# B&R Automation Studio project NAELD004C00R10L518F00 (part 5)

#### Act_Main_P0201.st
```iecst
(** 2018-12-21 **)
ACTION Act_Main_P0201:

	//Machine Bitmap //def70
	IF p_tyNtParamCurr.eProjMag = LDMagDual AND p_tyNtParamCurr.sJobNo = '2023-0258A01' THEN //AT&S
		tyP0201OpsTravLifter.tyOps.tyBitmapMc.uiValueIdx	:= 441-70;
	ELSIF p_tyNtParamCurr.eProjMag = LDMagDual AND p_tyNtParamCurr.sJobNo = '2023-0276A01' THEN //clarion
		tyP0201OpsTravLifter.tyOps.tyBitmapMc.uiValueIdx	:= 471-70;
	ELSIF p_tyNtParamCurr.eProjMag = LDMagDual AND p_tyNtParamCurr.bMagAutoVerifyPrep = TRUE THEN
		tyP0201OpsTravLifter.tyOps.tyBitmapMc.uiValueIdx	:= 200;//270
	ELSIF p_tyNtParamCurr.eProjMag = LDMagDual AND p_tyNtParamCurr.bMagAutoVerifyPrep = FALSE THEN
		tyP0201OpsTravLifter.tyOps.tyBitmapMc.uiValueIdx	:= 200;
	ELSIF p_tyNtParamCurr.eProjMag = LDMagTriple AND p_tyNtParamCurr.bProjLifterMagPlatform THEN
		tyP0201OpsTravLifter.tyOps.tyBitmapMc.uiValueIdx	:= 398-70;
	ELSIF p_tyNtParamCurr.eProjMag = LDMagTriple AND p_tyNtParamCurr.bProjLifterMagPlatform = FALSE AND p_tyNtParamCurr.bProjCurtainSenPrep THEN
		tyP0201OpsTravLifter.tyOps.tyBitmapMc.uiValueIdx	:= 361-70;
	ELSIF p_tyNtParamCurr.eProjMag = LDMagTriple THEN
		tyP0201OpsTravLifter.tyOps.tyBitmapMc.uiValueIdx	:= 3;
	ELSIF p_tyNtParamCurr.eProjMag = LDMagQuadruple THEN
		tyP0201OpsTravLifter.tyOps.tyBitmapMc.uiValueIdx	:= 7;
		fUIInRtStatOff(ADR(tyP0201OpsTravLifter.tyOps.tyLyrProdRear.uiRtStat));

	ELSE
		tyP0201OpsTravLifter.tyOps.tyBitmapMc.uiValueIdx	:= 0;
		fUIInRtStatHide(ADR(tyP0201OpsTravLifter.tyOps.tyLyrProdRear.uiRtStat));
	END_IF

	IF p_tyNtParamCurr.eProjMag <> LDMagQuadruple THEN
		fUIInRtStatHide(ADR(tyP0201OpsTravLifter.tyOps.tyLyrProdRear.uiRtStat));
	END_IF
		//Display
	tyP0201OpsTravLifter.tyOps.tyBtnToptoBtm.uiRtStat.0	:= TRUE;
	IF p_tyNtParamCurr.bProjLaneBPrep = FALSE THEN
		fUIInRtStatHide(ADR(tyP0201OpsTravLifter.tyIOMonitor.tyBtnDSBB.uiRtStat));

		fUIInRtStatHide(ADR(tyP0201OpsTravLifter.tyIOMonitor.tyBtnDBAB.uiRtStat));
	END_IF

	IF p_tyNtParamCurr.bProjInletShutPrep = FALSE THEN
		fUIInRtStatHide(ADR(tyP0201OpsTravLifter.tyIOMonitor.tyBtnInletShutterCloseSen.uiRtStat));
		fUIInRtStatHide(ADR(tyP0201OpsTravLifter.tyIOMonitor.tyBtnInletShutterOpenSen.uiRtStat));
		fUIInRtStatHide(ADR(tyP0201OpsTravLifter.tyIOMonitor.tyBtnInShutterCloseCtrl.uiRtStat));
		fUIInRtStatHide(ADR(tyP0201OpsTravLifter.tyIOMonitor.tyBtnInShutterOpenCtrl.uiRtStat));
	END_IF
	IF p_tyNtParamCurr.bProjShutter2Prep = FALSE THEN
		fUIInRtStatHide(ADR(tyP0201OpsTravLifter.tyIOMonitor.tyBtnInletShutterCloseSen2.uiRtStat));
		fUIInRtStatHide(ADR(tyP0201OpsTravLifter.tyIOMonitor.tyBtnInletShutterOpenSen2.uiRtStat));
		fUIInRtStatHide(ADR(tyP0201OpsTravLifter.tyIOMonitor.tyBtnInShutterCloseCtrl2.uiRtStat));
		fUIInRtStatHide(ADR(tyP0201OpsTravLifter.tyIOMonitor.tyBtnInShutterOpenCtrl2.uiRtStat));
	END_IF
	IF p_tyNtParamCurr.bProjShutter3Prep = FALSE THEN
		fUIInRtStatHide(ADR(tyP0201OpsTravLifter.tyIOMonitor.tyBtnInletShutterCloseSen3.uiRtStat));
		fUIInRtStatHide(ADR(tyP0201OpsTravLifter.tyIOMonitor.tyBtnInletShutterOpenSen3.uiRtStat));
		fUIInRtStatHide(ADR(tyP0201OpsTravLifter.tyIOMonitor.tyBtnInShutterCloseCtrl3.uiRtStat));
		fUIInRtStatHide(ADR(tyP0201OpsTravLifter.tyIOMonitor.tyBtnInShutterOpenCtrl3.uiRtStat));
	END_IF

	IF p_tyNtParamCurr.bProjOutletShutPrep = FALSE THEN
		fUIInRtStatHide(ADR(tyP0201OpsTravLifter.tyIOMonitor.tyBtnOutletShutterCloseSen.uiRtStat));
		fUIInRtStatHide(ADR(tyP0201OpsTravLifter.tyIOMonitor.tyBtnOutletShutterOpenSen.uiRtStat));
		fUIInRtStatHide(ADR(tyP0201OpsTravLifter.tyIOMonitor.tyBtnOutShutterCloseCtrl.uiRtStat));
		fUIInRtStatHide(ADR(tyP0201OpsTravLifter.tyIOMonitor.tyBtnOutShutterOpenCtrl.uiRtStat));
	END_IF
	IF p_tyNtParamCurr.bProjOutShutter2Prep = FALSE THEN
		fUIInRtStatHide(ADR(tyP0201OpsTravLifter.tyIOMonitor.tyBtnOutletShutterCloseSen2.uiRtStat));
		fUIInRtStatHide(ADR(tyP0201OpsTravLifter.tyIOMonitor.tyBtnOutletShutterOpenSen2.uiRtStat));
		fUIInRtStatHide(ADR(tyP0201OpsTravLifter.tyIOMonitor.tyBtnOutShutterCloseCtrl2.uiRtStat));
		fUIInRtStatHide(ADR(tyP0201OpsTravLifter.tyIOMonitor.tyBtnOutShutterOpenCtrl2.uiRtStat));
	END_IF

	//Change Parameter
	IF p_tyNtParamCurr.bProjLaneBPrep THEN
		tyP0201OpsTravLifter.tyParam.tyDrpDnMcMode.usiValueMaxIdx	:= 2;
	ELSE
		tyP0201OpsTravLifter.tyParam.tyDrpDnMcMode.usiValueMaxIdx	:= 0;
	END_IF

	//Motorised puller
	tyP0201OpsTravLifter.tyOps.tyNumPshrOffset.uiRtStat := NOT p_tyNtParamCurr.bAWPusherPrep;
	tyP0201OpsTravLifter.tyOps.tyNumMtrPshrExtSpd.uiRtStat := NOT p_tyNtParamCurr.bProjMotorizedPullerPrep;
	tyP0201OpsTravLifter.tyOps.tyNumMtrPshrExtTorq.uiRtStat := NOT p_tyNtParamCurr.bProjMotorizedPullerPrep;
	tyP0201OpsTravLifter.tyParam.tyNumPshrOffset.uiRtStat := NOT p_tyNtParamCurr.bAWPusherPrep;
	tyP0201OpsTravLifter.tyParam.tyNumMtrPshrExtSpd.uiRtStat := NOT p_tyNtParamCurr.bProjMotorizedPullerPrep;
	tyP0201OpsTravLifter.tyParam.tyNumMtrPshrExtTorq.uiRtStat := NOT p_tyNtParamCurr.bProjMotorizedPullerPrep;

	//Digital Input Used
	IF p_tyNtParamCurr.tyDISettings.diSafetyRlySig = 0 THEN
		fUIInRtStatHide(ADR(tyP0201OpsTravLifter.tyIOMonitor.tyBtnSafetyRlySig.uiRtStat));
	END_IF

	IF p_tyNtParamCurr.tyDISettings.diEStopSig = 0 THEN
		fUIInRtStatHide(ADR(tyP0201OpsTravLifter.tyIOMonitor.tyBtnEStop.uiRtStat));
	END_IF

	IF p_tyNtParamCurr.tyDISettings.diCoverSWSig = 0 THEN
		fUIInRtStatHide(ADR(tyP0201OpsTravLifter.tyIOMonitor.tyBtnCoverSWSig.uiRtStat));
	END_IF

	IF p_tyNtParamCurr.tyDISettings.diDSBA = 0 THEN
		fUIInRtStatHide(ADR(tyP0201OpsTravLifter.tyIOMonitor.tyBtnDSBA.uiRtStat));
	END_IF

	IF p_tyNtParamCurr.tyDISettings.diDSBB = 0 THEN
		fUIInRtStatHide(ADR(tyP0201OpsTravLifter.tyIOMonitor.tyBtnDSBB.uiRtStat));
	END_IF

	IF p_tyNtParamCurr.tyDISettings.diPullerExtRS = 0 THEN
		fUIInRtStatHide(ADR(tyP0201OpsTravLifter.tyIOMonitor.tyBtnPullerExtRS.uiRtStat));
	END_IF

	IF p_tyNtParamCurr.tyDISettings.diPullerRetRS = 0 THEN
		fUIInRtStatHide(ADR(tyP0201OpsTravLifter.tyIOMonitor.tyBtnPullerRetRS.uiRtStat));
	END_IF

	IF p_tyNtParamCurr.tyDISettings.diPullerRotHmRS = 0 THEN
		fUIInRtStatHide(ADR(tyP0201OpsTravLifter.tyIOMonitor.tyBtnPullerRotCylHmRS.uiRtStat));
	END_IF

	IF p_tyNtParamCurr.tyDISettings.diPullerRotRmRS = 0 THEN
		fUIInRtStatHide(ADR(tyP0201OpsTravLifter.tyIOMonitor.tyBtnPullerRotCylRmRS.uiRtStat));
	END_IF

	IF p_tyNtParamCurr.tyDISettings.diConvLftSen = 0 THEN
		fUIInRtStatHide(ADR(tyP0201OpsTravLifter.tyIOMonitor.tyBtnConvLftSen.uiRtStat));
	END_IF

	IF p_tyNtParamCurr.tyDISettings.diConvRgtSen = 0 THEN
		fUIInRtStatHide(ADR(tyP0201OpsTravLifter.tyIOMonitor.tyBtnConvRgtSen.uiRtStat));
	END_IF

	IF p_tyNtParamCurr.tyDISettings.diLifterTimingBeltSen = 0 THEN
		fUIInRtStatHide(ADR(tyP0201OpsTravLifter.tyIOMonitor.tyBtnLifterTmBeltSen.uiRtStat));
	END_IF

	IF p_tyNtParamCurr.tyDISettings.diLifterSafetyLmtSW1 = 0 THEN
		fUIInRtStatHide(ADR(tyP0201OpsTravLifter.tyIOMonitor.tyBtnLifterSafetyLmtSw1.uiRtStat));
	END_IF

	IF p_tyNtParamCurr.tyDISettings.diLifterSafetyLmtSW2 = 0 THEN
		fUIInRtStatHide(ADR(tyP0201OpsTravLifter.tyIOMonitor.tyBtnLifterSafetyLmtSw2.uiRtStat));
	END_IF

	IF p_tyNtParamCurr.tyDISettings.diInShutterOpenRS = 0 THEN
		fUIInRtStatHide(ADR(tyP0201OpsTravLifter.tyIOMonitor.tyBtnInletShutterOpenSen.uiRtStat));
	END_IF

	IF p_tyNtParamCurr.tyDISettings.diInShutterCloseRS = 0 THEN
		fUIInRtStatHide(ADR(tyP0201OpsTravLifter.tyIOMonitor.tyBtnInletShutterCloseSen.uiRtStat));
	END_IF

	IF p_tyNtParamCurr.tyDISettings.diOutShutterOpenRS = 0 THEN
		fUIInRtStatHide(ADR(tyP0201OpsTravLifter.tyIOMonitor.tyBtnOutletShutterOpenSen.uiRtStat));
	END_IF

	IF p_tyNtParamCurr.tyDISettings.diOutShutterCloseRS = 0 THEN
		fUIInRtStatHide(ADR(tyP0201OpsTravLifter.tyIOMonitor.tyBtnOutletShutterCloseSen.uiRtStat));
	END_IF

	IF p_tyNtParamCurr.tyDISettings.diPullerAntiJam = 0 THEN
		fUIInRtStatHide(ADR(tyP0201OpsTravLifter.tyIOMonitor.tyBtnAntiJamSen.uiRtStat));
	END_IF
	tyP0201OpsTravLifter.tyIOMonitor.tyBtnMagWidthChk.uiRtStat := p_tyNtParamCurr.tyDISettings.diMagWidthChkSen =0;

	//Digital Output Selected
	IF p_tyNtParamCurr.tyDOSettings.diSafetyRlyRst = 0 THEN
		fUIInRtStatHide(ADR(tyP0201OpsTravLifter.tyIOMonitor.tyBtnSafetyRlyRst.uiRtStat));
	END_IF

	IF p_tyNtParamCurr.tyDOSettings.diTLGreen = 0 THEN
		fUIInRtStatHide(ADR(tyP0201OpsTravLifter.tyIOMonitor.tyBtnTLGreen.uiRtStat));
	END_IF

	IF p_tyNtParamCurr.tyDOSettings.diTLAmber = 0 THEN
		fUIInRtStatHide(ADR(tyP0201OpsTravLifter.tyIOMonitor.tyBtnTLAmber.uiRtStat));
	ELSE
		IF p_tyNtParamCurr.eTLBuzMode = TLBuzModSiemens_2Colour THEN
			tyP0201OpsTravLifter.tyIOMonitor.tyBtnTLAmber.usiTxtIdx := 333-253; //253 amber
		END_IF
	END_IF

	IF p_tyNtParamCurr.tyDOSettings.diTLRed = 0 THEN
		fUIInRtStatHide(ADR(tyP0201OpsTravLifter.tyIOMonitor.tyBtnTLRed.uiRtStat));
	END_IF

	IF p_tyNtParamCurr.tyDOSettings.diBuzzer = 0 THEN
		fUIInRtStatHide(ADR(tyP0201OpsTravLifter.tyIOMonitor.tyBtnBuzzer.uiRtStat));
	END_IF

	IF p_tyNtParamCurr.tyDOSettings.diDBAA = 0 THEN
		fUIInRtStatHide(ADR(tyP0201OpsTravLifter.tyIOMonitor.tyBtnDBAA.uiRtStat));
	END_IF

	IF p_tyNtParamCurr.tyDOSettings.diDBAB = 0 THEN
		fUIInRtStatHide(ADR(tyP0201OpsTravLifter.tyIOMonitor.tyBtnDBAB.uiRtStat));
	END_IF

	IF p_tyNtParamCurr.tyDOSettings.diPullerExtCtrl = 0 THEN
		fUIInRtStatHide(ADR(tyP0201OpsTravLifter.tyIOMonitor.tyBtnPullerExtCtrl.uiRtStat));
	END_IF

	IF p_tyNtParamCurr.tyDOSettings.diPullerRetCtrl = 0 THEN
		fUIInRtStatHide(ADR(tyP0201OpsTravLifter.tyIOMonitor.tyBtnPullerRetCtrl.uiRtStat));
	END_IF

	IF p_tyNtParamCurr.tyDOSettings.diRotPullerCtrl = 0 THEN
		fUIInRtStatHide(ADR(tyP0201OpsTravLifter.tyIOMonitor.tyBtnRotPullerCtrl.uiRtStat));
	END_IF

	IF p_tyNtParamCurr.tyDOSettings.diInShutterOpenCtrl = 0 THEN
		fUIInRtStatHide(ADR(tyP0201OpsTravLifter.tyIOMonitor.tyBtnInShutterOpenCtrl.uiRtStat));
	END_IF

	IF p_tyNtParamCurr.tyDOSettings.diInShutterCloseCtrl = 0 THEN
		fUIInRtStatHide(ADR(tyP0201OpsTravLifter.tyIOMonitor.tyBtnInShutterCloseCtrl.uiRtStat));
	END_IF

	IF p_tyNtParamCurr.tyDOSettings.diOutShutterOpenCtrl = 0 THEN
		fUIInRtStatHide(ADR(tyP0201OpsTravLifter.tyIOMonitor.tyBtnOutShutterOpenCtrl.uiRtStat));
	END_IF

	IF p_tyNtParamCurr.tyDOSettings.diOutShutterCloseCtrl = 0 THEN
		fUIInRtStatHide(ADR(tyP0201OpsTravLifter.tyIOMonitor.tyBtnOutShutterCloseCtrl.uiRtStat));
	END_IF

	IF p_tyNtParamCurr.tyDOSettings.diPullConvMtrOn = 0 THEN
		fUIInRtStatHide(ADR(tyP0201OpsTravLifter.tyIOMonitor.tyBtnPullerConvMtrOn.uiRtStat));
	END_IF

	tyP0201OpsTravLifter.tyIOMonitor.tyBtnConvClrSen.uiRtStat := 	p_tyNtParamCurr.tyDISettings.diConvClrSen =0;
	tyP0201OpsTravLifter.tyIOMonitor.tyBtnUnlockSigDS.uiRtStat := 	p_tyNtParamCurr.tyDISettings.diDSUnlockCoverSig =0;
	tyP0201OpsTravLifter.tyIOMonitor.tyBtnSafetySigDS.uiRtStat := 	p_tyNtParamCurr.tyDISettings.diDSSafetySig =0;
	tyP0201OpsTravLifter.tyIOMonitor.tyBtnSftySglToUSDS.uiRtStat := 	p_tyNtParamCurr.tyDOSettings.diMcSafetySigToDS =0;

//	IF p_tyNtParamCurr.bLFProdWidth2Prep THEN
//		fUIInRtStatOff(ADR(tyP0201OpsTravLifter.tyOps.tyNumWidth2.uiRtStat));
//		fUIInRtStatHide(ADR(tyP0201OpsTravLifter.tyOps.tyNumWidth.uiRtStat));
//	ELSE
//		fUIInRtStatHide(ADR(tyP0201OpsTravLifter.tyOps.tyNumWidth2.uiRtStat));
//		fUIInRtStatOff(ADR(tyP0201OpsTravLifter.tyOps.tyNumWidth.uiRtStat));
//	END_IF
//
//	IF p_tyNtParamCurr.eProjMag = LDMagQuadruple THEN
//		fUIInRtStatOff(ADR(tyP0201OpsTravLifter.tyOps.tyNumWidth2.uiRtStat));
//		fUIInRtStatHide(ADR(tyP0201OpsTravLifter.tyOps.tyNumWidth.uiRtStat));
//	ELSE
		fUIInRtStatHide(ADR(tyP0201OpsTravLifter.tyOps.tyNumWidth2.uiRtStat));
		fUIInRtStatOff(ADR(tyP0201OpsTravLifter.tyOps.tyNumWidth.uiRtStat));
//	END_IF

END_ACTION
```

#### Act_Main_P0202.st
```iecst
(** 2018-12-21 **)
ACTION Act_Main_P0202:

	//Machine Bitmap//71

	IF p_tyNtParamCurr.eProjMag = LDMagDual AND p_tyNtParamCurr.sJobNo = '2023-0258A01' THEN //AT&S
		tyP0202OpsMag1.tyOps.tyBitmapMc.uiValueIdx	:= 442-71;
	ELSIF p_tyNtParamCurr.eProjMag = LDMagDual AND p_tyNtParamCurr.sJobNo = '2023-0276A01' THEN //clarion (RL)
		tyP0202OpsMag1.tyOps.tyBitmapMc.uiValueIdx	:= 472-71;
	ELSIF p_tyNtParamCurr.eProjMag = LDMagDual AND p_tyNtParamCurr.bMagAutoVerifyPrep = TRUE THEN
		tyP0202OpsMag1.tyOps.tyBitmapMc.uiValueIdx	:= 200;
	ELSIF p_tyNtParamCurr.eProjMag = LDMagDual AND p_tyNtParamCurr.bMagAutoVerifyPrep = FALSE THEN
		tyP0202OpsMag1.tyOps.tyBitmapMc.uiValueIdx	:= 200;
	ELSIF p_tyNtParamCurr.eProjMag = LDMagTriple AND p_tyNtParamCurr.bProjLifterMagPlatform THEN
		tyP0202OpsMag1.tyOps.tyBitmapMc.uiValueIdx	:= 399-71;
	ELSIF p_tyNtParamCurr.eProjMag = LDMagTriple AND p_tyNtParamCurr.bProjLifterMagPlatform =FALSE AND p_tyNtParamCurr.bProjCurtainSenPrep THEN
		tyP0202OpsMag1.tyOps.tyBitmapMc.uiValueIdx	:= 362-71;
	ELSIF p_tyNtParamCurr.eProjMag = LDMagTriple THEN
		tyP0202OpsMag1.tyOps.tyBitmapMc.uiValueIdx	:= 3;
	ELSIF p_tyNtParamCurr.eProjMag = LDMagQuadruple THEN
		tyP0202OpsMag1.tyOps.tyBitmapMc.uiValueIdx	:= 7;
	ELSE
		tyP0202OpsMag1.tyOps.tyBitmapMc.uiValueIdx	:= 0;
	END_IF

	//AIV
	tyP0202OpsMag1.tyOps.tyTxtLblAIV.uiRtStat.0		:= NOT p_tyNtParamCurr.bProjAGVPrep;
	tyP0202OpsMag1.tyOps.tyBtnAIVWifi.uiRtStat.0	:= NOT p_tyNtParamCurr.bProjAGVPrep;
	tyP0202OpsMag1.tyOps.tyBtnChgMag.uiRtStat.0		:= NOT(p_tyNtParamCurr.bProjAGVPrep AND p_tyNtParamCurr.bProjBtnInsertRmvMag);
	tyP0202OpsMag1.tyOps.tyBitmapChgMag.uiRtStat.0	:= NOT(p_tyNtParamCurr.bProjAGVPrep AND p_tyNtParamCurr.bProjBtnInsertRmvMag);

	//Motorized puller
	tyP0202OpsMag1.tyParam.tyNumPshrOffset.uiRtStat := NOT p_tyNtParamCurr.bAWPusherPrep;
	tyP0202OpsMag1.tyParam.tyNumMtrPshrExtSpd.uiRtStat := NOT p_tyNtParamCurr.bProjMotorizedPullerPrep;
	tyP0202OpsMag1.tyParam.tyNumMtrPshrExtTorq.uiRtStat := NOT p_tyNtParamCurr.bProjMotorizedPullerPrep;

	//Display
	IF p_tyNtParamCurr.bProjLaneBPrep = FALSE THEN
		fUIInRtStatHide(ADR(tyP0202OpsMag1.tyIOMonitor.tyBtnDSBB.uiRtStat));

		fUIInRtStatHide(ADR(tyP0202OpsMag1.tyIOMonitor.tyBtnDBAB.uiRtStat));
	END_IF
	tyP0202OpsMag1.tyOps.tyBtnToptoBtm.uiRtStat.0	:= TRUE;
	//Change Parameter
	IF p_tyNtParamCurr.bProjLaneBPrep THEN
		tyP0202OpsMag1.tyParam.tyDrpDnMcMode.usiValueMaxIdx	:= 2;
	ELSE
		tyP0202OpsMag1.tyParam.tyDrpDnMcMode.usiValueMaxIdx	:= 0;
	END_IF

	//Digital Input Used
	IF p_tyNtParamCurr.tyDISettings.diSafetyRlySig = 0 THEN
		fUIInRtStatHide(ADR(tyP0202OpsMag1.tyIOMonitor.tyBtnSafetyRlySig.uiRtStat));
	END_IF

	IF p_tyNtParamCurr.tyDISettings.diEStopSig = 0 THEN
		fUIInRtStatHide(ADR(tyP0202OpsMag1.tyIOMonitor.tyBtnEStop.uiRtStat));
	END_IF

	IF p_tyNtParamCurr.tyDISettings.diCoverSWSig = 0 THEN
		fUIInRtStatHide(ADR(tyP0202OpsMag1.tyIOMonitor.tyBtnCoverSWSig.uiRtStat));
	END_IF

	IF p_tyNtParamCurr.tyDISettings.diDSBA = 0 THEN
		fUIInRtStatHide(ADR(tyP0202OpsMag1.tyIOMonitor.tyBtnDSBA.uiRtStat));
	END_IF

	IF p_tyNtParamCurr.tyDISettings.diDSBB = 0 THEN
		fUIInRtStatHide(ADR(tyP0202OpsMag1.tyIOMonitor.tyBtnDSBB.uiRtStat));
	END_IF

	IF p_tyNtParamCurr.tyDISettings.diMag1FixedClampRS = 0 THEN
		fUIInRtStatHide(ADR(tyP0202OpsMag1.tyIOMonitor.tyBtnMag1FixedClmpRS.uiRtStat));
	END_IF

	IF p_tyNtParamCurr.tyDISettings.diMag1FixedUnclampRS = 0 THEN
		fUIInRtStatHide(ADR(tyP0202OpsMag1.tyIOMonitor.tyBtnMag1FixedUnclmpRS.uiRtStat));
	END_IF

	IF p_tyNtParamCurr.tyDISettings.diMag1RemoteClampRS = 0 THEN
		fUIInRtStatHide(ADR(tyP0202OpsMag1.tyIOMonitor.tyBtnMag1RmtClmpRS.uiRtStat));
	END_IF

	IF p_tyNtParamCurr.tyDISettings.diMag1RemoteUnclampRS = 0 THEN
		fUIInRtStatHide(ADR(tyP0202OpsMag1.tyIOMonitor.tyBtnMag1RmtUnclmpRS.uiRtStat));
	END_IF

	IF p_tyNtParamCurr.tyDISettings.diMagConvEntSen1 = 0 THEN
		fUIInRtStatHide(ADR(tyP0202OpsMag1.tyIOMonitor.tyBtnMag1ConvEntrySen.uiRtStat));
	END_IF

	IF p_tyNtParamCurr.tyDISettings.diMagPresentSen1 = 0 THEN
		fUIInRtStatHide(ADR(tyP0202OpsMag1.tyIOMonitor.tyBtnMag1PresentSen.uiRtStat));
	END_IF

	IF p_tyNtParamCurr.tyDISettings.diMag1AGVInPosSen1 = 0 THEN
		fUIInRtStatHide(ADR(tyP0202OpsMag1.tyIOMonitor.tyBtnMag1AIVInPosSen1.uiRtStat));
	END_IF

	IF p_tyNtParamCurr.tyDISettings.diMag1AGVInPosSen2 = 0 THEN
		fUIInRtStatHide(ADR(tyP0202OpsMag1.tyIOMonitor.tyBtnMag1AIVInPosSen2.uiRtStat));
	END_IF

	IF p_tyNtParamCurr.tyDISettings.diMag1OrientChkSen1 = 0 THEN
		fUIInRtStatHide(ADR(tyP0202OpsMag1.tyIOMonitor.tyBtnMag1OrientationChkSen1.uiRtStat));
	END_IF

	IF p_tyNtParamCurr.tyDISettings.diMag1OrientChkSen2 = 0 THEN
		fUIInRtStatHide(ADR(tyP0202OpsMag1.tyIOMonitor.tyBtnMag1OrientationChkSen2.uiRtStat));
	END_IF

	tyP0202OpsMag1.tyIOMonitor.tyBtnMagDetSen.uiRtStat.0			:= p_tyNtParamCurr.tyDISettings.diMag1FixedSideDetect = 0;
	tyP0202OpsMag1.tyIOMonitor.tyBtnTrllyExtRS.uiRtStat.0			:= p_tyNtParamCurr.tyDISettings.diTrolleyExtRS1 = 0;
	tyP0202OpsMag1.tyIOMonitor.tyBtnTrllyPresentSen.uiRtStat.0		:= p_tyNtParamCurr.tyDISettings.diTrolleyPreSen1 = 0;
	tyP0202OpsMag1.tyIOMonitor.tyBtnSltLckSen.uiRtStat.0			:= p_tyNtParamCurr.tyDISettings.diSlotLckSenMag1 = 0;

	//Digital Output Selected
	IF p_tyNtParamCurr.tyDOSettings.diSafetyRlyRst = 0 THEN
		fUIInRtStatHide(ADR(tyP0202OpsMag1.tyIOMonitor.tyBtnSafetyRlyRst.uiRtStat));
	END_IF

	IF p_tyNtParamCurr.tyDOSettings.diTLGreen = 0 THEN
		fUIInRtStatHide(ADR(tyP0202OpsMag1.tyIOMonitor.tyBtnTLGreen.uiRtStat));
	END_IF

	IF p_tyNtParamCurr.tyDOSettings.diTLAmber = 0 THEN
		fUIInRtStatHide(ADR(tyP0202OpsMag1.tyIOMonitor.tyBtnTLAmber.uiRtStat));
	ELSE
		IF p_tyNtParamCurr.eTLBuzMode = TLBuzModSiemens_2Colour THEN
			tyP0202OpsMag1.tyIOMonitor.tyBtnTLAmber.usiTxtIdx := 333-253; //253 amber
		END_IF
	END_IF

	IF p_tyNtParamCurr.tyDOSettings.diTLRed = 0 THEN
		fUIInRtStatHide(ADR(tyP0202OpsMag1.tyIOMonitor.tyBtnTLRed.uiRtStat));
	END_IF

	IF p_tyNtParamCurr.tyDOSettings.diBuzzer = 0 THEN
		fUIInRtStatHide(ADR(tyP0202OpsMag1.tyIOMonitor.tyBtnBuzzer.uiRtStat));
	END_IF

	IF p_tyNtParamCurr.tyDOSettings.diDBAA = 0 THEN
		fUIInRtStatHide(ADR(tyP0202OpsMag1.tyIOMonitor.tyBtnDBAA.uiRtStat));
	END_IF

	IF p_tyNtParamCurr.tyDOSettings.diDBAB = 0 THEN
		fUIInRtStatHide(ADR(tyP0202OpsMag1.tyIOMonitor.tyBtnDBAB.uiRtStat));
	END_IF

	IF p_tyNtParamCurr.tyDOSettings.diMag1FixedClampCtrl = 0 THEN
		fUIInRtStatHide(ADR(tyP0202OpsMag1.tyIOMonitor.tyBtnMag1FixedClampCtrl.uiRtStat));
	END_IF

	IF p_tyNtParamCurr.tyDOSettings.diMag1FixedClampOpenCtrl = 0 THEN //KS
		fUIInRtStatHide(ADR(tyP0202OpsMag1.tyIOMonitor.tyBtnMag1FixedClampCtrl.uiRtStat));
	END_IF

	IF p_tyNtParamCurr.tyDOSettings.diMag1RemoteClampCtrl = 0 THEN
		fUIInRtStatHide(ADR(tyP0202OpsMag1.tyIOMonitor.tyBtnMag1RemoteClampCtrl.uiRtStat));
	END_IF

	IF p_tyNtParamCurr.tyDOSettings.diMag1RemoteClampOpenCtrl = 0 THEN //KS
		fUIInRtStatHide(ADR(tyP0202OpsMag1.tyIOMonitor.tyBtnMag1RemoteClampCtrl.uiRtStat));
	END_IF

	IF p_tyNtParamCurr.tyDOSettings.diMag1ConvMtrIn = 0 THEN
		fUIInRtStatHide(ADR(tyP0202OpsMag1.tyIOMonitor.tyBtnMag1ConvMtrIn.uiRtStat));
	END_IF

	IF p_tyNtParamCurr.tyDOSettings.diMag1ConvMtrOut = 0 THEN
		fUIInRtStatHide(ADR(tyP0202OpsMag1.tyIOMonitor.tyBtnMag1ConvMtrOut.uiRtStat));
	END_IF
	tyP0202OpsMag1.tyIOMonitor.tyBtnTrllyExtCtrl.uiRtStat.0			:= p_tyNtParamCurr.tyDOSettings.diTrolleyLckCtrl1 = 0;

	tyP0202OpsMag1.tyIOMonitor.tyBtnMagSelClampCtrl.uiRtStat.0		:= NOT p_tyNtParamCurr.bMagAutoVerifyPrep;
	tyP0202OpsMag1.tyIOMonitor.tyBtnHeightSen.uiRtStat.0			:= NOT (p_tyNtParamCurr.bMagAutoVerifyPrep OR p_tyNtParamCurr.bProjMagHeightChkPrep);
	tyP0202OpsMag1.tyIOMonitor.tyBtnCAB717Sen.uiRtStat.0			:= NOT p_tyNtParamCurr.bMagAutoVerifyPrep;
	tyP0202OpsMag1.tyIOMonitor.tyBtnMagLargeSen.uiRtStat.0			:= NOT p_tyNtParamCurr.bMagAutoVerifyPrep;
	tyP0202OpsMag1.tyIOMonitor.tyBtnMagSmallSen.uiRtStat.0			:= NOT p_tyNtParamCurr.bMagAutoVerifyPrep;
	tyP0202OpsMag1.tyIOMonitor.tyBtnSelUnclampRS.uiRtStat.0			:= NOT p_tyNtParamCurr.bMagAutoVerifyPrep;

//	IF p_tyNtParamCurr.eProjMag = LDMagQuadruple THEN
//		fUIInRtStatOff(ADR(tyP0202OpsMag1.tyOps.tyNumWidth2.uiRtStat));
//		fUIInRtStatHide(ADR(tyP0202OpsMag1.tyOps.tyNumWidth.uiRtStat));
//	ELSE
		fUIInRtStatHide(ADR(tyP0202OpsMag1.tyOps.tyNumWidth2.uiRtStat));
		fUIInRtStatOff(ADR(tyP0202OpsMag1.tyOps.tyNumWidth.uiRtStat));
//	END_IF

	tyP0202OpsMag1.tyOps.tyBtnUnloadMag.uiRtStat.0 := NOT p_tyNtParamCurr.bProjLifterMagPlatform;
	tyP0202OpsMag1.tyOps.tyBitmapUnloadMag.uiRtStat.0 := NOT p_tyNtParamCurr.bProjLifterMagPlatform;
	tyP0202OpsMag1.tyOps.tyBtnChgMag.uiRtStat.0 := p_tyNtParamCurr.bProjLifterMagPlatform;

END_ACTION
```

#### Act_Main_P0203.st
```iecst
(** 2018-12-21 **)
ACTION Act_Main_P0203:

	//Machine Bitmap//72
	IF p_tyNtParamCurr.eProjMag = LDMagDual AND p_tyNtParamCurr.sJobNo = '2023-0258A01' THEN //AT&S
		tyP0203OpsMag2.tyOps.tyBitmapMc.uiValueIdx	:= 443-72;
	ELSIF p_tyNtParamCurr.eProjMag = LDMagDual AND p_tyNtParamCurr.sJobNo = '2023-0276A01' THEN //clarion (RL)
		tyP0203OpsMag2.tyOps.tyBitmapMc.uiValueIdx	:= 473-72;
	ELSIF p_tyNtParamCurr.eProjMag = LDMagDual AND p_tyNtParamCurr.bMagAutoVerifyPrep = TRUE THEN
		tyP0203OpsMag2.tyOps.tyBitmapMc.uiValueIdx	:= 200;
	ELSIF p_tyNtParamCurr.eProjMag = LDMagDual AND p_tyNtParamCurr.bMagAutoVerifyPrep = FALSE THEN
		tyP0203OpsMag2.tyOps.tyBitmapMc.uiValueIdx	:= 200;
	ELSIF p_tyNtParamCurr.eProjMag = LDMagTriple AND p_tyNtParamCurr.bProjLifterMagPlatform THEN
		tyP0203OpsMag2.tyOps.tyBitmapMc.uiValueIdx	:= 400-72;
	ELSIF p_tyNtParamCurr.eProjMag = LDMagTriple AND p_tyNtParamCurr.bProjLifterMagPlatform =FALSE AND p_tyNtParamCurr.bProjCurtainSenPrep THEN
		tyP0203OpsMag2.tyOps.tyBitmapMc.uiValueIdx	:= 363-72;
	ELSIF p_tyNtParamCurr.eProjMag = LDMagTriple THEN
		tyP0203OpsMag2.tyOps.tyBitmapMc.uiValueIdx	:= 3;
	ELSIF p_tyNtParamCurr.eProjMag = LDMagQuadruple THEN
		tyP0203OpsMag2.tyOps.tyBitmapMc.uiValueIdx	:= 7;
	ELSE
		tyP0203OpsMag2.tyOps.tyBitmapMc.uiValueIdx	:= 0;
	END_IF

	//AIV
	tyP0203OpsMag2.tyOps.tyTxtLblAIV.uiRtStat.0		:= NOT p_tyNtParamCurr.bProjAGVPrep;
	tyP0203OpsMag2.tyOps.tyBtnAIVWifi.uiRtStat.0	:= NOT p_tyNtParamCurr.bProjAGVPrep;
	tyP0203OpsMag2.tyOps.tyBtnChgMag.uiRtStat.0		:= NOT(p_tyNtParamCurr.bProjAGVPrep AND p_tyNtParamCurr.bProjBtnInsertRmvMag);
	tyP0203OpsMag2.tyOps.tyBitmapChgMag.uiRtStat.0	:= NOT(p_tyNtParamCurr.bProjAGVPrep AND p_tyNtParamCurr.bProjBtnInsertRmvMag);

	//Motorized puller
	tyP0203OpsMag2.tyParam.tyNumPshrOffset.uiRtStat := NOT p_tyNtParamCurr.bAWPusherPrep;
	tyP0203OpsMag2.tyParam.tyNumMtrPshrExtSpd.uiRtStat := NOT p_tyNtParamCurr.bProjMotorizedPullerPrep;
	tyP0203OpsMag2.tyParam.tyNumMtrPshrExtTorq.uiRtStat := NOT p_tyNtParamCurr.bProjMotorizedPullerPrep;

	//Display
	IF p_tyNtParamCurr.bProjLaneBPrep = FALSE THEN
		fUIInRtStatHide(ADR(tyP0203OpsMag2.tyIOMonitor.tyBtnDSBB.uiRtStat));

		fUIInRtStatHide(ADR(tyP0203OpsMag2.tyIOMonitor.tyBtnDBAB.uiRtStat));
	END_IF
	tyP0203OpsMag2.tyOps.tyBtnToptoBtm.uiRtStat.0	:= TRUE;
	//Change Parameter
	IF p_tyNtParamCurr.bProjLaneBPrep THEN
		tyP0203OpsMag2.tyParam.tyDrpDnMcMode.usiValueMaxIdx	:= 2;
	ELSE
		tyP0203OpsMag2.tyParam.tyDrpDnMcMode.usiValueMaxIdx	:= 0;
	END_IF

	//Digital Input Used
	IF p_tyNtParamCurr.tyDISettings.diSafetyRlySig = 0 THEN
		fUIInRtStatHide(ADR(tyP0203OpsMag2.tyIOMonitor.tyBtnSafetyRlySig.uiRtStat));
	END_IF

	IF p_tyNtParamCurr.tyDISettings.diEStopSig = 0 THEN
		fUIInRtStatHide(ADR(tyP0203OpsMag2.tyIOMonitor.tyBtnEStop.uiRtStat));
	END_IF

	IF p_tyNtParamCurr.tyDISettings.diCoverSWSig = 0 THEN
		fUIInRtStatHide(ADR(tyP0203OpsMag2.tyIOMonitor.tyBtnCoverSWSig.uiRtStat));
	END_IF

	IF p_tyNtParamCurr.tyDISettings.diDSBA = 0 THEN
		fUIInRtStatHide(ADR(tyP0203OpsMag2.tyIOMonitor.tyBtnDSBA.uiRtStat));
	END_IF

	IF p_tyNtParamCurr.tyDISettings.diDSBB = 0 THEN
		fUIInRtStatHide(ADR(tyP0203OpsMag2.tyIOMonitor.tyBtnDSBB.uiRtStat));
	END_IF

	IF p_tyNtParamCurr.tyDISettings.diMag2FixedClampRS = 0 THEN
		fUIInRtStatHide(ADR(tyP0203OpsMag2.tyIOMonitor.tyBtnMag2FixedClmpRS.uiRtStat));
	END_IF

	IF p_tyNtParamCurr.tyDISettings.diMag2FixedUnclampRS = 0 THEN
		fUIInRtStatHide(ADR(tyP0203OpsMag2.tyIOMonitor.tyBtnMag2FixedUnclmpRS.uiRtStat));
	END_IF

	IF p_tyNtParamCurr.tyDISettings.diMag2RemoteClampRS = 0 THEN
		fUIInRtStatHide(ADR(tyP0203OpsMag2.tyIOMonitor.tyBtnMag2RmtClmpRS.uiRtStat));
	END_IF

	IF p_tyNtParamCurr.tyDISettings.diMag2RemoteUnclampRS = 0 THEN
		fUIInRtStatHide(ADR(tyP0203OpsMag2.tyIOMonitor.tyBtnMag2RmtUnclmpRS.uiRtStat));
	END_IF

	IF p_tyNtParamCurr.tyDISettings.diMagConvEntSen2 = 0 THEN
		fUIInRtStatHide(ADR(tyP0203OpsMag2.tyIOMonitor.tyBtnMag2ConvEntrySen.uiRtStat));
	END_IF

	IF p_tyNtParamCurr.tyDISettings.diMagPresentSen2 = 0 THEN
		fUIInRtStatHide(ADR(tyP0203OpsMag2.tyIOMonitor.tyBtnMag2PresentSen.uiRtStat));
	END_IF

	IF p_tyNtParamCurr.tyDISettings.diMag2AGVInPosSen1 = 0 THEN
		fUIInRtStatHide(ADR(tyP0203OpsMag2.tyIOMonitor.tyBtnMag2AIVInPosSen1.uiRtStat));
	END_IF

	IF p_tyNtParamCurr.tyDISettings.diMag2AGVInPosSen2 = 0 THEN
		fUIInRtStatHide(ADR(tyP0203OpsMag2.tyIOMonitor.tyBtnMag2AIVInPosSen2.uiRtStat));
	END_IF

	IF p_tyNtParamCurr.tyDISettings.diMag1OrientChkSen1 = 0 THEN
		fUIInRtStatHide(ADR(tyP0203OpsMag2.tyIOMonitor.tyBtnMag2OrientationChkSen1.uiRtStat));
	END_IF

	IF p_tyNtParamCurr.tyDISettings.diMag2OrientChkSen2 = 0 THEN
		fUIInRtStatHide(ADR(tyP0203OpsMag2.tyIOMonitor.tyBtnMag2OrientationChkSen2.uiRtStat));
	END_IF
	tyP0203OpsMag2.tyIOMonitor.tyBtnMagDetSen.uiRtStat.0			:= p_tyNtParamCurr.tyDISettings.diMag2FixedSideDetect = 0;
	tyP0203OpsMag2.tyIOMonitor.tyBtnTrllyExtRS.uiRtStat.0			:= p_tyNtParamCurr.tyDISettings.diTrolleyExtRS2 = 0;
	tyP0203OpsMag2.tyIOMonitor.tyBtnTrllyPresentSen.uiRtStat.0		:= p_tyNtParamCurr.tyDISettings.diTrolleyPreSen2 = 0;
	tyP0203OpsMag2.tyIOMonitor.tyBtnSltLckSen.uiRtStat.0			:= p_tyNtParamCurr.tyDISettings.diSlotLckSenMag2 = 0;

	//Digital Output Selected
	IF p_tyNtParamCurr.tyDOSettings.diSafetyRlyRst = 0 THEN
		fUIInRtStatHide(ADR(tyP0203OpsMag2.tyIOMonitor.tyBtnSafetyRlyRst.uiRtStat));
	END_IF

	IF p_tyNtParamCurr.tyDOSettings.diTLGreen = 0 THEN
		fUIInRtStatHide(ADR(tyP0203OpsMag2.tyIOMonitor.tyBtnTLGreen.uiRtStat));
	END_IF

	IF p_tyNtParamCurr.tyDOSettings.diTLAmber = 0 THEN
		fUIInRtStatHide(ADR(tyP0203OpsMag2.tyIOMonitor.tyBtnTLAmber.uiRtStat));
	ELSE
		IF p_tyNtParamCurr.eTLBuzMode = TLBuzModSiemens_2Colour THEN
			tyP0203OpsMag2.tyIOMonitor.tyBtnTLAmber.usiTxtIdx := 333-253; //253 amber
		END_IF
	END_IF

	IF p_tyNtParamCurr.tyDOSettings.diTLRed = 0 THEN
		fUIInRtStatHide(ADR(tyP0203OpsMag2.tyIOMonitor.tyBtnTLRed.uiRtStat));
	END_IF

	IF p_tyNtParamCurr.tyDOSettings.diBuzzer = 0 THEN
		fUIInRtStatHide(ADR(tyP0203OpsMag2.tyIOMonitor.tyBtnBuzzer.uiRtStat));
	END_IF

	IF p_tyNtParamCurr.tyDOSettings.diDBAA = 0 THEN
		fUIInRtStatHide(ADR(tyP0203OpsMag2.tyIOMonitor.tyBtnDBAA.uiRtStat));
	END_IF

	IF p_tyNtParamCurr.tyDOSettings.diDBAB = 0 THEN
		fUIInRtStatHide(ADR(tyP0203OpsMag2.tyIOMonitor.tyBtnDBAB.uiRtStat));
	END_IF

	IF p_tyNtParamCurr.tyDOSettings.diMag2FixedClampCtrl = 0 THEN
		fUIInRtStatHide(ADR(tyP0203OpsMag2.tyIOMonitor.tyBtnMag2FixedClampCtrl.uiRtStat));
	END_IF

	IF p_tyNtParamCurr.tyDOSettings.diMag2RemoteClampCtrl = 0 THEN
		fUIInRtStatHide(ADR(tyP0203OpsMag2.tyIOMonitor.tyBtnMag2RemoteClampCtrl.uiRtStat));
	END_IF

	IF p_tyNtParamCurr.tyDOSettings.diMag2ConvMtrIn = 0 THEN
		fUIInRtStatHide(ADR(tyP0203OpsMag2.tyIOMonitor.tyBtnMag2ConvMtrIn.uiRtStat));
	END_IF

	IF p_tyNtParamCurr.tyDOSettings.diMag2ConvMtrOut = 0 THEN
		fUIInRtStatHide(ADR(tyP0203OpsMag2.tyIOMonitor.tyBtnMag2ConvMtrOut.uiRtStat));
	END_IF
	tyP0203OpsMag2.tyIOMonitor.tyBtnTrllyExtCtrl.uiRtStat.0			:= p_tyNtParamCurr.tyDOSettings.diTrolleyLckCtrl2 = 0;

	tyP0203OpsMag2.tyIOMonitor.tyBtnMagSelClampCtrl.uiRtStat.0		:= NOT p_tyNtParamCurr.bMagAutoVerifyPrep;
	tyP0203OpsMag2.tyIOMonitor.tyBtnHeightSen.uiRtStat.0			:= NOT (p_tyNtParamCurr.bMagAutoVerifyPrep OR p_tyNtParamCurr.bProjMagHeightChkPrep);
	tyP0203OpsMag2.tyIOMonitor.tyBtnCAB717Sen.uiRtStat.0			:= NOT p_tyNtParamCurr.bMagAutoVerifyPrep;
	tyP0203OpsMag2.tyIOMonitor.tyBtnMagLargeSen.uiRtStat.0			:= NOT p_tyNtParamCurr.bMagAutoVerifyPrep;
	tyP0203OpsMag2.tyIOMonitor.tyBtnMagSmallSen.uiRtStat.0			:= NOT p_tyNtParamCurr.bMagAutoVerifyPrep;
	tyP0203OpsMag2.tyIOMonitor.tyBtnSelUnclampRS.uiRtStat.0			:= NOT p_tyNtParamCurr.bMagAutoVerifyPrep;

//	IF p_tyNtParamCurr.eProjMag = LDMagQuadruple THEN
//		fUIInRtStatOff(ADR(tyP0203OpsMag2.tyOps.tyNumWidth2.uiRtStat));
//		fUIInRtStatHide(ADR(tyP0203OpsMag2.tyOps.tyNumWidth.uiRtStat));
//	ELSE
		fUIInRtStatHide(ADR(tyP0203OpsMag2.tyOps.tyNumWidth2.uiRtStat));
		fUIInRtStatOff(ADR(tyP0203OpsMag2.tyOps.tyNumWidth.uiRtStat));
//	END_IF

	tyP0203OpsMag2.tyOps.tyBtnUnloadMag.uiRtStat.0 := NOT p_tyNtParamCurr.bProjLifterMagPlatform;
	tyP0203OpsMag2.tyOps.tyBitmapUnloadMag.uiRtStat.0 := NOT p_tyNtParamCurr.bProjLifterMagPlatform;
	tyP0203OpsMag2.tyOps.tyBtnChgMag.uiRtStat.0 := p_tyNtParamCurr.bProjLifterMagPlatform;

END_ACTION
```

#### Act_Main_P0204.st
```iecst
(** 2021-05-31 **)
ACTION Act_Main_P0204:

	//Machine Bitmap//73

	IF p_tyNtParamCurr.eProjMag = LDMagDual AND p_tyNtParamCurr.bMagAutoVerifyPrep = TRUE THEN
		tyP0204OpsMag3.tyOps.tyBitmapMc.uiValueIdx	:= 200;//273
	ELSIF p_tyNtParamCurr.eProjMag = LDMagDual AND p_tyNtParamCurr.bMagAutoVerifyPrep = FALSE THEN
		tyP0204OpsMag3.tyOps.tyBitmapMc.uiValueIdx	:= 200;
	ELSIF p_tyNtParamCurr.eProjMag = LDMagTriple AND p_tyNtParamCurr.bProjLifterMagPlatform THEN
		tyP0204OpsMag3.tyOps.tyBitmapMc.uiValueIdx	:= 401-73;
	ELSIF p_tyNtParamCurr.eProjMag = LDMagTriple AND p_tyNtParamCurr.bProjLifterMagPlatform =FALSE AND p_tyNtParamCurr.bProjCurtainSenPrep THEN
		tyP0204OpsMag3.tyOps.tyBitmapMc.uiValueIdx	:= 364-73;
	ELSIF p_tyNtParamCurr.eProjMag = LDMagTriple THEN
		tyP0204OpsMag3.tyOps.tyBitmapMc.uiValueIdx	:= 3;
	ELSIF p_tyNtParamCurr.eProjMag = LDMagQuadruple THEN
		tyP0204OpsMag3.tyOps.tyBitmapMc.uiValueIdx	:= 7;
	ELSE
		tyP0204OpsMag3.tyOps.tyBitmapMc.uiValueIdx	:= 0;
	END_IF

	//AIV
	tyP0204OpsMag3.tyOps.tyTxtLblAIV.uiRtStat.0		:= NOT p_tyNtParamCurr.bProjAGVPrep;
	tyP0204OpsMag3.tyOps.tyBtnAIVWifi.uiRtStat.0	:= NOT p_tyNtParamCurr.bProjAGVPrep;
	tyP0204OpsMag3.tyOps.tyBtnChgMag.uiRtStat.0		:= NOT(p_tyNtParamCurr.bProjAGVPrep AND p_tyNtParamCurr.bProjBtnInsertRmvMag);
	tyP0204OpsMag3.tyOps.tyBitmapChgMag.uiRtStat.0	:= NOT(p_tyNtParamCurr.bProjAGVPrep AND p_tyNtParamCurr.bProjBtnInsertRmvMag);

	//Motorized puller
	tyP0204OpsMag3.tyParam.tyNumPshrOffset.uiRtStat := NOT p_tyNtParamCurr.bAWPusherPrep;
	tyP0204OpsMag3.tyParam.tyNumMtrPshrExtSpd.uiRtStat := NOT p_tyNtParamCurr.bProjMotorizedPullerPrep;
	tyP0204OpsMag3.tyParam.tyNumMtrPshrExtTorq.uiRtStat := NOT p_tyNtParamCurr.bProjMotorizedPullerPrep;

	//Display
	IF p_tyNtParamCurr.bProjLaneBPrep = FALSE THEN
		fUIInRtStatHide(ADR(tyP0204OpsMag3.tyIOMonitor.tyBtnDSBB.uiRtStat));

		fUIInRtStatHide(ADR(tyP0204OpsMag3.tyIOMonitor.tyBtnDBAB.uiRtStat));
	END_IF
	tyP0204OpsMag3.tyOps.tyBtnToptoBtm.uiRtStat.0	:= TRUE;
	//Change Parameter
	IF p_tyNtParamCurr.bProjLaneBPrep THEN
		tyP0204OpsMag3.tyParam.tyDrpDnMcMode.usiValueMaxIdx	:= 2;
	ELSE
		tyP0204OpsMag3.tyParam.tyDrpDnMcMode.usiValueMaxIdx	:= 0;
	END_IF

	//Digital Input Used
	IF p_tyNtParamCurr.tyDISettings.diSafetyRlySig = 0 THEN
		fUIInRtStatHide(ADR(tyP0204OpsMag3.tyIOMonitor.tyBtnSafetyRlySig.uiRtStat));
	END_IF

	IF p_tyNtParamCurr.tyDISettings.diEStopSig = 0 THEN
		fUIInRtStatHide(ADR(tyP0204OpsMag3.tyIOMonitor.tyBtnEStop.uiRtStat));
	END_IF

	IF p_tyNtParamCurr.tyDISettings.diCoverSWSig = 0 THEN
		fUIInRtStatHide(ADR(tyP0204OpsMag3.tyIOMonitor.tyBtnCoverSWSig.uiRtStat));
	END_IF

	IF p_tyNtParamCurr.tyDISettings.diDSBA = 0 THEN
		fUIInRtStatHide(ADR(tyP0204OpsMag3.tyIOMonitor.tyBtnDSBA.uiRtStat));
	END_IF

	IF p_tyNtParamCurr.tyDISettings.diDSBB = 0 THEN
		fUIInRtStatHide(ADR(tyP0204OpsMag3.tyIOMonitor.tyBtnDSBB.uiRtStat));
	END_IF

	IF p_tyNtParamCurr.tyDISettings.diMag3FixedClampRS = 0 THEN
		fUIInRtStatHide(ADR(tyP0204OpsMag3.tyIOMonitor.tyBtnMag3FixedClmpRS.uiRtStat));
	END_IF

	IF p_tyNtParamCurr.tyDISettings.diMag3FixedUnclampRS = 0 THEN
		fUIInRtStatHide(ADR(tyP0204OpsMag3.tyIOMonitor.tyBtnMag3FixedUnclmpRS.uiRtStat));
	END_IF

	IF p_tyNtParamCurr.tyDISettings.diMag3RemoteClampRS = 0 THEN
		fUIInRtStatHide(ADR(tyP0204OpsMag3.tyIOMonitor.tyBtnMag3RmtClmpRS.uiRtStat));
	END_IF

	IF p_tyNtParamCurr.tyDISettings.diMag3RemoteUnclampRS = 0 THEN
		fUIInRtStatHide(ADR(tyP0204OpsMag3.tyIOMonitor.tyBtnMag3RmtUnclmpRS.uiRtStat));
	END_IF

	IF p_tyNtParamCurr.tyDISettings.diMagConvEntSen3 = 0 THEN
		fUIInRtStatHide(ADR(tyP0204OpsMag3.tyIOMonitor.tyBtnMag3ConvEntrySen.uiRtStat));
	END_IF

	IF p_tyNtParamCurr.tyDISettings.diMagPresentSen3 = 0 THEN
		fUIInRtStatHide(ADR(tyP0204OpsMag3.tyIOMonitor.tyBtnMag3PresentSen.uiRtStat));
	END_IF

	IF p_tyNtParamCurr.tyDISettings.diMag3AGVInPosSen1 = 0 THEN
		fUIInRtStatHide(ADR(tyP0204OpsMag3.tyIOMonitor.tyBtnMag3AIVInPosSen1.uiRtStat));
	END_IF

	IF p_tyNtParamCurr.tyDISettings.diMag3AGVInPosSen2 = 0 THEN
		fUIInRtStatHide(ADR(tyP0204OpsMag3.tyIOMonitor.tyBtnMag3AIVInPosSen2.uiRtStat));
	END_IF

	IF p_tyNtParamCurr.tyDISettings.diMag3OrientChkSen1 = 0 THEN
		fUIInRtStatHide(ADR(tyP0204OpsMag3.tyIOMonitor.tyBtnMag3OrientationChkSen1.uiRtStat));
	END_IF

	IF p_tyNtParamCurr.tyDISettings.diMag3OrientChkSen2 = 0 THEN
		fUIInRtStatHide(ADR(tyP0204OpsMag3.tyIOMonitor.tyBtnMag3OrientationChkSen2.uiRtStat));
	END_IF
	tyP0204OpsMag3.tyIOMonitor.tyBtnMagDetSen.uiRtStat.0			:= p_tyNtParamCurr.tyDISettings.diMag3FixedSideDetect = 0;

	//Digital Output Selected
	IF p_tyNtParamCurr.tyDOSettings.diSafetyRlyRst = 0 THEN
		fUIInRtStatHide(ADR(tyP0204OpsMag3.tyIOMonitor.tyBtnSafetyRlyRst.uiRtStat));
	END_IF

	IF p_tyNtParamCurr.tyDOSettings.diTLGreen = 0 THEN
		fUIInRtStatHide(ADR(tyP0204OpsMag3.tyIOMonitor.tyBtnTLGreen.uiRtStat));
	END_IF

	IF p_tyNtParamCurr.tyDOSettings.diTLAmber = 0 THEN
		fUIInRtStatHide(ADR(tyP0204OpsMag3.tyIOMonitor.tyBtnTLAmber.uiRtStat));
	ELSE
		IF p_tyNtParamCurr.eTLBuzMode = TLBuzModSiemens_2Colour THEN
			tyP0204OpsMag3.tyIOMonitor.tyBtnTLAmber.usiTxtIdx := 333-253; //253 amber
		END_IF
	END_IF

	IF p_tyNtParamCurr.tyDOSettings.diTLRed = 0 THEN
		fUIInRtStatHide(ADR(tyP0204OpsMag3.tyIOMonitor.tyBtnTLRed.uiRtStat));
	END_IF

	IF p_tyNtParamCurr.tyDOSettings.diBuzzer = 0 THEN
		fUIInRtStatHide(ADR(tyP0203OpsMag2.tyIOMonitor.tyBtnBuzzer.uiRtStat));
	END_IF

	IF p_tyNtParamCurr.tyDOSettings.diDBAA = 0 THEN
		fUIInRtStatHide(ADR(tyP0203OpsMag2.tyIOMonitor.tyBtnDBAA.uiRtStat));
	END_IF

	IF p_tyNtParamCurr.tyDOSettings.diDBAB = 0 THEN
		fUIInRtStatHide(ADR(tyP0203OpsMag2.tyIOMonitor.tyBtnDBAB.uiRtStat));
	END_IF

	IF p_tyNtParamCurr.tyDOSettings.diMag3FixedClampCtrl = 0 THEN
		fUIInRtStatHide(ADR(tyP0204OpsMag3.tyIOMonitor.tyBtnMag3FixedClampCtrl.uiRtStat));
	END_IF

	IF p_tyNtParamCurr.tyDOSettings.diMag3RemoteClampCtrl = 0 THEN
		fUIInRtStatHide(ADR(tyP0204OpsMag3.tyIOMonitor.tyBtnMag3RemoteClampCtrl.uiRtStat));
	END_IF

	IF p_tyNtParamCurr.tyDOSettings.diMag3ConvMtrIn = 0 THEN
		fUIInRtStatHide(ADR(tyP0204OpsMag3.tyIOMonitor.tyBtnMag3ConvMtrIn.uiRtStat));
	END_IF

	IF p_tyNtParamCurr.tyDOSettings.diMag3ConvMtrOut = 0 THEN
		fUIInRtStatHide(ADR(tyP0204OpsMag3.tyIOMonitor.tyBtnMag3ConvMtrOut.uiRtStat));
	END_IF

	tyP0204OpsMag3.tyIOMonitor.tyBtnMagSelClampCtrl.uiRtStat.0		:= NOT p_tyNtParamCurr.bMagAutoVerifyPrep;
	tyP0204OpsMag3.tyIOMonitor.tyBtnHeightSen.uiRtStat.0			:= NOT (p_tyNtParamCurr.bMagAutoVerifyPrep OR p_tyNtParamCurr.bProjMagHeightChkPrep);
	tyP0204OpsMag3.tyIOMonitor.tyBtnCAB717Sen.uiRtStat.0			:= NOT p_tyNtParamCurr.bMagAutoVerifyPrep;
	tyP0204OpsMag3.tyIOMonitor.tyBtnMagLargeSen.uiRtStat.0			:= NOT p_tyNtParamCurr.bMagAutoVerifyPrep;
	tyP0204OpsMag3.tyIOMonitor.tyBtnMagSmallSen.uiRtStat.0			:= NOT p_tyNtParamCurr.bMagAutoVerifyPrep;
	tyP0204OpsMag3.tyIOMonitor.tyBtnSelUnclampRS.uiRtStat.0			:= NOT p_tyNtParamCurr.bMagAutoVerifyPrep;

//	IF p_tyNtParamCurr.eProjMag = LDMagQuadruple THEN
//		fUIInRtStatOff(ADR(tyP0204OpsMag3.tyOps.tyNumWidth2.uiRtStat));
//		fUIInRtStatHide(ADR(tyP0204OpsMag3.tyOps.tyNumWidth.uiRtStat));
//	ELSE
		fUIInRtStatHide(ADR(tyP0204OpsMag3.tyOps.tyNumWidth2.uiRtStat));
		fUIInRtStatOff(ADR(tyP0204OpsMag3.tyOps.tyNumWidth.uiRtStat));
//	END_IF

	tyP0204OpsMag3.tyOps.tyBtnUnloadMag.uiRtStat.0 := NOT p_tyNtParamCurr.bProjLifterMagPlatform;
	tyP0204OpsMag3.tyOps.tyBitmapUnloadMag.uiRtStat.0 := NOT p_tyNtParamCurr.bProjLifterMagPlatform;
	tyP0204OpsMag3.tyOps.tyBtnChgMag.uiRtStat.0 := p_tyNtParamCurr.bProjLifterMagPlatform;

END_ACTION
```

#### Act_Main_P0205.st
```iecst
(** 2021-05-14 **)
ACTION Act_Main_P0205:

	//Machine Bitmap
	IF p_tyNtParamCurr.eProjMag = LDMagDual THEN
		tyP0205OpsAIV.tyIOMonitor.tyBitmapMc.usiValueIdx	:= 217;
		fUIInRtStatOff(ADR(tyP0205OpsAIV.tyIOMonitor.tyLyr12.uiRtStat));
		fUIInRtStatHide(ADR(tyP0205OpsAIV.tyIOMonitor.tyLyr3.uiRtStat));
		fUIInRtStatHide(ADR(tyP0205OpsAIV.tyIOMonitor.tyLyr4.uiRtStat));
	ELSIF p_tyNtParamCurr.eProjMag = LDMagTriple THEN
		tyP0205OpsAIV.tyIOMonitor.tyBitmapMc.usiValueIdx	:= 215;
		fUIInRtStatHide(ADR(tyP0205OpsAIV.tyIOMonitor.tyLyr12.uiRtStat));
		fUIInRtStatOff(ADR(tyP0205OpsAIV.tyIOMonitor.tyLyr3.uiRtStat));
		fUIInRtStatHide(ADR(tyP0205OpsAIV.tyIOMonitor.tyLyr4.uiRtStat));

	ELSIF p_tyNtParamCurr.eProjMag = LDMagQuadruple THEN
		tyP0205OpsAIV.tyIOMonitor.tyBitmapMc.usiValueIdx	:= 216;
		fUIInRtStatHide(ADR(tyP0205OpsAIV.tyIOMonitor.tyLyr12.uiRtStat));
		fUIInRtStatHide(ADR(tyP0205OpsAIV.tyIOMonitor.tyLyr3.uiRtStat));
		fUIInRtStatOff(ADR(tyP0205OpsAIV.tyIOMonitor.tyLyr4.uiRtStat));
	END_IF

	tyP0205OpsAIV.tyIOMonitor.tyBtnAIVSotRCVOk1.uiRtStat.0 := NOT(p_tyNtParamCurr.bProjSOTSensorPrep);
	tyP0205OpsAIV.tyIOMonitor.tyBtnAIVSotRCVOk2.uiRtStat.0 := NOT(p_tyNtParamCurr.bProjSOTSensorPrep);
	tyP0205OpsAIV.tyIOMonitor.tyBtnAIVSotRCVOk3.uiRtStat.0 := NOT(p_tyNtParamCurr.bProjSOTSensorPrep);
	tyP0205OpsAIV.tyIOMonitor.tyBtnAIVSotRCVOk4.uiRtStat.0 := NOT(p_tyNtParamCurr.bProjSOTSensorPrep);

	tyP0205OpsAIV.tyIOMonitor.tyStringMesName.uiRtStat.0 := NOT(p_tyNtParamCurr.bShowMESName);
	IF p_tyNtParamCurr.bShowFMorMESActive THEN
		tyP0205OpsAIV.tyIOMonitor.tyBtnMESActive.usiTxtIdx := 17;//Fleet management active
	ELSE
		tyP0205OpsAIV.tyIOMonitor.tyBtnMESActive.usiTxtIdx := 0;//Mes active
	END_IF

	//Siemens 3LD
	tyP0205OpsAIV.tyIOMonitor.tyBtnReqAIVToBring1.uiRtStat := TRUE;//p_tyNtParamCurr.eCustomerReq = Siemens OR p_tyNtParamCurr.eCustomerReq = We_Fabricate;
	tyP0205OpsAIV.tyIOMonitor.tyBtnReqAIVToGet1.uiRtStat := TRUE;//p_tyNtParamCurr.eCustomerReq = Siemens OR p_tyNtParamCurr.eCustomerReq = We_Fabricate;
	tyP0205OpsAIV.tyIOMonitor.tyBtnReqAIVToBring2.uiRtStat := TRUE;//p_tyNtParamCurr.eCustomerReq = Siemens OR p_tyNtParamCurr.eCustomerReq = We_Fabricate;
	tyP0205OpsAIV.tyIOMonitor.tyBtnReqAIVToGet2.uiRtStat := TRUE;//p_tyNtParamCurr.eCustomerReq = Siemens OR p_tyNtParamCurr.eCustomerReq = We_Fabricate;
	tyP0205OpsAIV.tyIOMonitor.tyBtnReqAIVToBring3.uiRtStat := TRUE;//p_tyNtParamCurr.eCustomerReq = Siemens OR p_tyNtParamCurr.eCustomerReq = We_Fabricate;
	tyP0205OpsAIV.tyIOMonitor.tyBtnReqAIVToGet3.uiRtStat := TRUE;//p_tyNtParamCurr.eCustomerReq = Siemens OR p_tyNtParamCurr.eCustomerReq = We_Fabricate;

END_ACTION
```

#### Act_Main_P0206.st
```iecst
(** 2018-12-21 **)
ACTION Act_Main_P0206:

	//Machine Bitmap
	tyP0206OpsMag4.tyOps.tyBitmapMc.usiValueIdx	:= 0;

	//AIV
	tyP0206OpsMag4.tyOps.tyTxtLblAIV.uiRtStat.0		:= NOT p_tyNtParamCurr.bProjAGVPrep;
	tyP0206OpsMag4.tyOps.tyBtnAIVWifi.uiRtStat.0	:= NOT p_tyNtParamCurr.bProjAGVPrep;
	tyP0206OpsMag4.tyOps.tyBtnChgMag.uiRtStat.0		:= NOT(p_tyNtParamCurr.bProjAGVPrep AND p_tyNtParamCurr.bProjBtnInsertRmvMag);
	tyP0206OpsMag4.tyOps.tyBitmapChgMag.uiRtStat.0	:= NOT(p_tyNtParamCurr.bProjAGVPrep AND p_tyNtParamCurr.bProjBtnInsertRmvMag);

	//Display
	IF p_tyNtParamCurr.bProjLaneBPrep = FALSE THEN
		fUIInRtStatHide(ADR(tyP0206OpsMag4.tyIOMonitor.tyBtnDSBB.uiRtStat));

		fUIInRtStatHide(ADR(tyP0206OpsMag4.tyIOMonitor.tyBtnDBAB.uiRtStat));
	END_IF
	tyP0206OpsMag4.tyOps.tyBtnToptoBtm.uiRtStat.0	:= TRUE;
	//Change Parameter
	IF p_tyNtParamCurr.bProjLaneBPrep THEN
		tyP0206OpsMag4.tyParam.tyDrpDnMcMode.usiValueMaxIdx	:= 2;
	ELSE
		tyP0206OpsMag4.tyParam.tyDrpDnMcMode.usiValueMaxIdx	:= 0;
	END_IF

	//Digital Input Used
	IF p_tyNtParamCurr.tyDISettings.diSafetyRlySig = 0 THEN
		fUIInRtStatHide(ADR(tyP0206OpsMag4.tyIOMonitor.tyBtnSafetyRlySig.uiRtStat));
	END_IF

	IF p_tyNtParamCurr.tyDISettings.diEStopSig = 0 THEN
		fUIInRtStatHide(ADR(tyP0206OpsMag4.tyIOMonitor.tyBtnEStop.uiRtStat));
	END_IF

	IF p_tyNtParamCurr.tyDISettings.diCoverSWSig = 0 THEN
		fUIInRtStatHide(ADR(tyP0206OpsMag4.tyIOMonitor.tyBtnCoverSWSig.uiRtStat));
	END_IF

	IF p_tyNtParamCurr.tyDISettings.diDSBA = 0 THEN
		fUIInRtStatHide(ADR(tyP0206OpsMag4.tyIOMonitor.tyBtnDSBA.uiRtStat));
	END_IF

	IF p_tyNtParamCurr.tyDISettings.diDSBB = 0 THEN
		fUIInRtStatHide(ADR(tyP0206OpsMag4.tyIOMonitor.tyBtnDSBB.uiRtStat));
	END_IF

	IF p_tyNtParamCurr.tyDISettings.diMag4FixedClampRS = 0 THEN
		fUIInRtStatHide(ADR(tyP0206OpsMag4.tyIOMonitor.tyBtnMag4FixedClmpRS.uiRtStat));
	END_IF

	IF p_tyNtParamCurr.tyDISettings.diMag4FixedUnclampRS = 0 THEN
		fUIInRtStatHide(ADR(tyP0206OpsMag4.tyIOMonitor.tyBtnMag4FixedUnclmpRS.uiRtStat));
	END_IF

	IF p_tyNtParamCurr.tyDISettings.diMag4RemoteClampRS = 0 THEN
		fUIInRtStatHide(ADR(tyP0206OpsMag4.tyIOMonitor.tyBtnMag4RmtClmpRS.uiRtStat));
	END_IF

	IF p_tyNtParamCurr.tyDISettings.diMag4RemoteUnclampRS = 0 THEN
		fUIInRtStatHide(ADR(tyP0206OpsMag4.tyIOMonitor.tyBtnMag4RmtUnclmpRS.uiRtStat));
	END_IF

	IF p_tyNtParamCurr.tyDISettings.diMagConvEntSen4 = 0 THEN
		fUIInRtStatHide(ADR(tyP0206OpsMag4.tyIOMonitor.tyBtnMag4ConvEntrySen.uiRtStat));
	END_IF

	IF p_tyNtParamCurr.tyDISettings.diMagPresentSen4 = 0 THEN
		fUIInRtStatHide(ADR(tyP0206OpsMag4.tyIOMonitor.tyBtnMag4PresentSen.uiRtStat));
	END_IF

	IF p_tyNtParamCurr.tyDISettings.diMag4AGVInPosSen1 = 0 THEN
		fUIInRtStatHide(ADR(tyP0206OpsMag4.tyIOMonitor.tyBtnMag4AIVInPosSen1.uiRtStat));
	END_IF

	IF p_tyNtParamCurr.tyDISettings.diMag4AGVInPosSen2 = 0 THEN
		fUIInRtStatHide(ADR(tyP0206OpsMag4.tyIOMonitor.tyBtnMag4AIVInPosSen2.uiRtStat));
	END_IF

	IF p_tyNtParamCurr.tyDISettings.diMag4OrientChkSen1 = 0 THEN
		fUIInRtStatHide(ADR(tyP0206OpsMag4.tyIOMonitor.tyBtnMag4OrientationChkSen1.uiRtStat));
	END_IF

	IF p_tyNtParamCurr.tyDISettings.diMag4OrientChkSen2 = 0 THEN
		fUIInRtStatHide(ADR(tyP0206OpsMag4.tyIOMonitor.tyBtnMag4OrientationChkSen2.uiRtStat));
	END_IF

	//Digital Output Selected
	IF p_tyNtParamCurr.tyDOSettings.diSafetyRlyRst = 0 THEN
		fUIInRtStatHide(ADR(tyP0206OpsMag4.tyIOMonitor.tyBtnSafetyRlyRst.uiRtStat));
	END_IF

	IF p_tyNtParamCurr.tyDOSettings.diTLGreen = 0 THEN
		fUIInRtStatHide(ADR(tyP0206OpsMag4.tyIOMonitor.tyBtnTLGreen.uiRtStat));
	END_IF

	IF p_tyNtParamCurr.tyDOSettings.diTLAmber = 0 THEN
		fUIInRtStatHide(ADR(tyP0206OpsMag4.tyIOMonitor.tyBtnTLAmber.uiRtStat));
	END_IF

	IF p_tyNtParamCurr.tyDOSettings.diTLRed = 0 THEN
		fUIInRtStatHide(ADR(tyP0206OpsMag4.tyIOMonitor.tyBtnTLRed.uiRtStat));
	END_IF

	IF p_tyNtParamCurr.tyDOSettings.diBuzzer = 0 THEN
		fUIInRtStatHide(ADR(tyP0206OpsMag4.tyIOMonitor.tyBtnBuzzer.uiRtStat));
	END_IF

	IF p_tyNtParamCurr.tyDOSettings.diDBAA = 0 THEN
		fUIInRtStatHide(ADR(tyP0206OpsMag4.tyIOMonitor.tyBtnDBAA.uiRtStat));
	END_IF

	IF p_tyNtParamCurr.tyDOSettings.diDBAB = 0 THEN
		fUIInRtStatHide(ADR(tyP0206OpsMag4.tyIOMonitor.tyBtnDBAB.uiRtStat));
	END_IF

	IF p_tyNtParamCurr.tyDOSettings.diMag4FixedClampCtrl = 0 THEN
		fUIInRtStatHide(ADR(tyP0206OpsMag4.tyIOMonitor.tyBtnMag4FixedClampCtrl.uiRtStat));
	END_IF

	IF p_tyNtParamCurr.tyDOSettings.diMag4RemoteClampCtrl = 0 THEN
		fUIInRtStatHide(ADR(tyP0206OpsMag4.tyIOMonitor.tyBtnMag4RemoteClampCtrl.uiRtStat));
	END_IF

	IF p_tyNtParamCurr.tyDOSettings.diMag4ConvMtrIn = 0 THEN
		fUIInRtStatHide(ADR(tyP0206OpsMag4.tyIOMonitor.tyBtnMag4ConvMtrIn.uiRtStat));
	END_IF

	IF p_tyNtParamCurr.tyDOSettings.diMag4ConvMtrOut = 0 THEN
		fUIInRtStatHide(ADR(tyP0206OpsMag4.tyIOMonitor.tyBtnMag4ConvMtrOut.uiRtStat));
	END_IF

	tyP0206OpsMag4.tyIOMonitor.tyBtnMagSelClampCtrl.uiRtStat.0		:= NOT p_tyNtParamCurr.bMagAutoVerifyPrep;
	tyP0206OpsMag4.tyIOMonitor.tyBtnHeightSen.uiRtStat.0			:= NOT p_tyNtParamCurr.bMagAutoVerifyPrep;
	tyP0206OpsMag4.tyIOMonitor.tyBtnCAB717Sen.uiRtStat.0			:= NOT p_tyNtParamCurr.bMagAutoVerifyPrep;
	tyP0206OpsMag4.tyIOMonitor.tyBtnMagLargeSen.uiRtStat.0			:= NOT p_tyNtParamCurr.bMagAutoVerifyPrep;
	tyP0206OpsMag4.tyIOMonitor.tyBtnMagSmallSen.uiRtStat.0			:= NOT p_tyNtParamCurr.bMagAutoVerifyPrep;
	tyP0206OpsMag4.tyIOMonitor.tyBtnSelUnclampRS.uiRtStat.0			:= NOT p_tyNtParamCurr.bMagAutoVerifyPrep;

//	IF p_tyNtParamCurr.eProjMag = LDMagQuadruple THEN
//		fUIInRtStatOff(ADR(tyP0206OpsMag4.tyOps.tyNumWidth2.uiRtStat));
//		fUIInRtStatHide(ADR(tyP0206OpsMag4.tyOps.tyNumWidth.uiRtStat));
//	ELSE
		fUIInRtStatHide(ADR(tyP0206OpsMag4.tyOps.tyNumWidth2.uiRtStat));
		fUIInRtStatOff(ADR(tyP0206OpsMag4.tyOps.tyNumWidth.uiRtStat));
//	END_IF

	tyP0206OpsMag4.tyOps.tyBtnUnloadMag.uiRtStat.0 := NOT p_tyNtParamCurr.bProjLifterMagPlatform;
	tyP0206OpsMag4.tyOps.tyBitmapUnloadMag.uiRtStat.0 := NOT p_tyNtParamCurr.bProjLifterMagPlatform;
	tyP0206OpsMag4.tyOps.tyBtnChgMag.uiRtStat.0 := p_tyNtParamCurr.bProjLifterMagPlatform;

END_ACTION
```

#### Act_Main_P0400.st
```iecst
ACTION Act_Main_P0400:

	//Product Selection
	tyP0400ProdSel.tyProdSel.tyStringRecipeNm.sValue		:= p_tyProdRcpCurrRcp0.sRcpNm;
	tyP0400ProdSel.tyProdSel.tyNumProdWidth.diValue			:= p_tyProdRcpCurrRcp0.diWidthInUM;
	tyP0400ProdSel.tyProdSel.tyNumMaxSlt.diValue			:= p_tyProdRcpCurrRcp0.diMaxSltValue;
	tyP0400ProdSel.tyProdSel.tyNumMinSlt.diValue			:= p_tyProdRcpCurrRcp0.diMinSltValue;
	tyP0400ProdSel.tyProdSel.tyNumPitch.diValue				:= p_tyProdRcpCurrRcp0.diPitch;
	tyP0400ProdSel.tyProdSel.tyBtnToptoBtm.bValue			:= p_tyProdRcpCurrRcp0.bTopToBtm;
	tyP0400ProdSel.tyProdSel.tyBtnLongBrd.bValue			:= p_tyProdRcpCurrRcp0.bLongBrd;
	tyP0400ProdSel.tyProdSel.tyTxtMcMode.usiValueIdx		:= p_tyProdRcpCurrRcp0.usiMcMod;
	tyP0400ProdSel.tyProdSel.tyTxtFlippedBrd.usiValueIdx	:= p_tyProdRcpCurrRcp0.usiFlippedBrd;

	tyP0400ProdSel.tyProdSel.tyNumProdWidthRear.diValue		:= p_tyProdRcpCurrRcp0.diWidthInUMRear;
	tyP0400ProdSel.tyProdSel.tyNumPitchRear.diValue			:= p_tyProdRcpCurrRcp0.diPitchRear;
	tyP0400ProdSel.tyProdSel.tyNumMinSltRear.diValue		:= p_tyProdRcpCurrRcp0.diMinSltValueRear;
	tyP0400ProdSel.tyProdSel.tyNumMaxSltRear.diValue		:= p_tyProdRcpCurrRcp0.diMaxSltValueRear;
	tyP0400ProdSel.tyProdSel.tyNumPshrOffset.diValue		:= p_tyProdRcpCurrRcp0.diPshrOffset;

	tyP0400ProdSel.tyProdSel.tyTxtFlippedBrd.uiRtStat.0	:= TRUE;
	tyP0400ProdSel.tyProdSel.tyBtnToptoBtm.uiRtStat.0	:= TRUE;
	tyP0400ProdSel.tyRcpDet.tyBtnToptoBtm.uiRtStat.0	:= TRUE;

	IF p_tyNtParamCurr.bLFProdWidth2Prep THEN
		fUIInRtStatOff(ADR(tyP0400ProdSel.tyProdSel.tyNumProdWidth2.uiRtStat));
		fUIInRtStatHide(ADR(tyP0400ProdSel.tyProdSel.tyNumProdWidth.uiRtStat));

		fUIInRtStatOff(ADR(tyP0400ProdSel.tyRcpDet.tyNumProdWidth2.uiRtStat));
		fUIInRtStatHide(ADR(tyP0400ProdSel.tyRcpDet.tyNumProdWidth.uiRtStat));

		tyP0400ProdSel.tyProdSel.tyTableRecipe.tyStringTitle2Col2Row0.sValue:= 'US | DS Width';

	ELSE
		fUIInRtStatHide(ADR(tyP0400ProdSel.tyProdSel.tyNumProdWidth2.uiRtStat));
		fUIInRtStatOff(ADR(tyP0400ProdSel.tyProdSel.tyNumProdWidth.uiRtStat));

		fUIInRtStatHide(ADR(tyP0400ProdSel.tyRcpDet.tyNumProdWidth2.uiRtStat));
		fUIInRtStatOff(ADR(tyP0400ProdSel.tyRcpDet.tyNumProdWidth.uiRtStat));

		tyP0400ProdSel.tyProdSel.tyTableRecipe.tyStringTitle2Col2Row0.sValue:= 'Product Width';
	END_IF

	CASE p_tyNtParamCurr.eProjMag OF
		LDMagDual, LDMagTriple:
			fUIInRtStatOff(ADR(tyP0400ProdSel.tyProdSel.tyNotQuadrupleLyr.uiRtStat));
			fUIInRtStatHide(ADR(tyP0400ProdSel.tyProdSel.tyQuadrupleLyr.uiRtStat));

		LDMagQuadruple:
			fUIInRtStatHide(ADR(tyP0400ProdSel.tyProdSel.tyNotQuadrupleLyr.uiRtStat));
			fUIInRtStatOff(ADR(tyP0400ProdSel.tyProdSel.tyQuadrupleLyr.uiRtStat));
	END_CASE

	//Motorized Pusher
	tyP0400ProdSel.tyProdSel.tyTxtMtrPshrExtSpd.uiRtStat.0	:= NOT p_tyNtParamCurr.bProjMotorizedPullerPrep;
	tyP0400ProdSel.tyProdSel.tyTxtMtrPshrExtTorq.uiRtStat.0	:= NOT p_tyNtParamCurr.bProjMotorizedPullerPrep;
	tyP0400ProdSel.tyProdSel.tyNumMtrPshrExtSpd.uiRtStat.0	:= NOT p_tyNtParamCurr.bProjMotorizedPullerPrep;
	tyP0400ProdSel.tyProdSel.tyNumMtrPshrExtTorq.uiRtStat.0	:= NOT p_tyNtParamCurr.bProjMotorizedPullerPrep;
	tyP0400ProdSel.tyRcpDet.tyTxtMtrPshrExtSpd.uiRtStat.0	:= NOT p_tyNtParamCurr.bProjMotorizedPullerPrep;
	tyP0400ProdSel.tyRcpDet.tyTxtMtrPshrExtTorq.uiRtStat.0	:= NOT p_tyNtParamCurr.bProjMotorizedPullerPrep;
	tyP0400ProdSel.tyRcpDet.tyNumMtrPshrExtSpd.uiRtStat.0	:= NOT p_tyNtParamCurr.bProjMotorizedPullerPrep;
	tyP0400ProdSel.tyRcpDet.tyNumMtrPshrExtTorq.uiRtStat.0	:= NOT p_tyNtParamCurr.bProjMotorizedPullerPrep;
	tyP0400ProdSel.tyProdSel.tyNumMtrPshrExtSpd.diValue		:= p_tyProdRcpCurrRcp0.diMtrPshrExtSpd;
	tyP0400ProdSel.tyProdSel.tyNumMtrPshrExtTorq.diValue	:= p_tyProdRcpCurrRcp0.diMtrPshrExtTorq;

	//Puller Offset
	tyP0400ProdSel.tyProdSel.tyNumPshrOffset.uiRtStat.0		:= NOT p_tyNtParamCurr.bAWPusherPrep;
	tyP0400ProdSel.tyProdSel.tyTxtPshrOffset.uiRtStat.0		:= NOT p_tyNtParamCurr.bAWPusherPrep;
	tyP0400ProdSel.tyRcpDet.tyNumPshrOffset.uiRtStat.0		:= NOT p_tyNtParamCurr.bAWPusherPrep;
	tyP0400ProdSel.tyRcpDet.tyTxtPshrOffset.uiRtStat.0		:= NOT p_tyNtParamCurr.bAWPusherPrep;

END_ACTION
```

#### Act_Main_P0410.st
```iecst
ACTION Act_Main_P0410:

	//Display
	tyP0410MagSel.tyMagSel.tyTxtLifMag3Slt1PosLbl.uiRtStat.0	:= NOT(p_tyNtParamCurr.eProjMag = LDMagTriple OR p_tyNtParamCurr.eProjMag = LDMagQuadruple);
	tyP0410MagSel.tyMagSel.tyNumLifterMag3Slt1Pos.uiRtStat.0	:= NOT(p_tyNtParamCurr.eProjMag = LDMagTriple OR p_tyNtParamCurr.eProjMag = LDMagQuadruple);

	tyP0410MagSel.tyMagDet.tyTxtLifMag3Slt1PosLbl.uiRtStat.0	:= NOT(p_tyNtParamCurr.eProjMag = LDMagTriple OR p_tyNtParamCurr.eProjMag = LDMagQuadruple);
	tyP0410MagSel.tyMagDet.tyNumLifterMag3Slt1Pos.uiRtStat.0	:= NOT(p_tyNtParamCurr.eProjMag = LDMagTriple OR p_tyNtParamCurr.eProjMag = LDMagQuadruple);

	tyP0410MagSel.tyMagSel.tyTxtTravPosMag3Lbl.uiRtStat.0	:= NOT(p_tyNtParamCurr.eProjMag = LDMagTriple OR p_tyNtParamCurr.eProjMag = LDMagQuadruple);
	tyP0410MagSel.tyMagSel.tyNumTravPosMag3.uiRtStat.0		:= NOT(p_tyNtParamCurr.eProjMag = LDMagTriple OR p_tyNtParamCurr.eProjMag = LDMagQuadruple);

	tyP0410MagSel.tyMagDet.tyTxtTravPosMag3Lbl.uiRtStat.0	:= NOT(p_tyNtParamCurr.eProjMag = LDMagTriple OR p_tyNtParamCurr.eProjMag = LDMagQuadruple);
	tyP0410MagSel.tyMagDet.tyNumTravPosMag3.uiRtStat.0		:= NOT(p_tyNtParamCurr.eProjMag = LDMagTriple OR p_tyNtParamCurr.eProjMag = LDMagQuadruple);

	//Magazine Selection
	tyP0410MagSel.tyMagSel.tyStringRecipeNm.sValue			:= p_tyMagRcpCurrRcp.sRcpNm;
	tyP0410MagSel.tyMagSel.tyNumMaxSlt.diValue				:= p_tyMagRcpCurrRcp.diTtlSlt;
	tyP0410MagSel.tyMagSel.tyNumSltToSltDist.diValue		:= p_tyMagRcpCurrRcp.diSltToSltInUM;
	tyP0410MagSel.tyMagSel.tyNumLifterMag1Slt1Pos.diValue	:= p_tyMagRcpCurrRcp.diMag1Slt1PosInUM;
	tyP0410MagSel.tyMagSel.tyNumLifterMag2Slt1Pos.diValue	:= p_tyMagRcpCurrRcp.diMag2Slt1PosInUM;
	tyP0410MagSel.tyMagSel.tyNumLifterMag3Slt1Pos.diValue	:= p_tyMagRcpCurrRcp.diMag3Slt1PosInUM;
	tyP0410MagSel.tyMagSel.tyNumLifterMag4Slt1Pos.diValue	:= p_tyMagRcpCurrRcp.diMag4Slt1PosInUM;
	tyP0410MagSel.tyMagSel.tyNumTravPosMag1.diValue			:= p_tyMagRcpCurrRcp.diMag1TravPosInUM;
	tyP0410MagSel.tyMagSel.tyNumTravPosMag2.diValue			:= p_tyMagRcpCurrRcp.diMag2TravPosInUM;
	tyP0410MagSel.tyMagSel.tyNumTravPosMag3.diValue			:= p_tyMagRcpCurrRcp.diMag3TravPosInUM;
	tyP0410MagSel.tyMagSel.tyNumTravPosMag4.diValue			:= p_tyMagRcpCurrRcp.diMag4TravPosInUM;
	tyP0410MagSel.tyMagSel.tyTxtMagModel.usiValueIdx		:= p_tyMagRcpCurrRcp.usiMagModel;
	tyP0410MagSel.tyMagSel.tyNumMagMaxBrdWidth.diValue		:= p_tyMagRcpCurrRcp.diMagMaxBrdWidth;

	tyP0410MagSel.tyMagSel.tyNumLifterMag4Slt1Pos.uiRtStat.0	:= NOT(p_tyNtParamCurr.eProjMag = LDMagQuadruple);
	tyP0410MagSel.tyMagSel.tyNumTravPosMag4.uiRtStat.0		:= NOT(p_tyNtParamCurr.eProjMag = LDMagQuadruple);

	tyP0410MagSel.tyMagSel.tyBtnSafetyBar.uiRtStat.0	:= NOT(p_tyNtParamCurr.bProjMagSafetyBarPrep);
	tyP0410MagSel.tyMagDet.tyBtnSafetyBar.uiRtStat.0	:= NOT(p_tyNtParamCurr.bProjMagSafetyBarPrep);

	tyP0410MagSel.tyMagDet.tyNumLifterMag4Slt1Pos.uiRtStat.0	:= NOT(p_tyNtParamCurr.eProjMag = LDMagQuadruple);
	tyP0410MagSel.tyMagDet.tyNumTravPosMag4.uiRtStat.0		:= NOT(p_tyNtParamCurr.eProjMag = LDMagQuadruple);

	tyP0410MagSel.tyMagSel.tyTxtMagTitle.usiValueIdx	:= 0;

	tyP0410MagSel.tyMagSel.tyBtnMagHeightChkEn.uiRtStat.0	:= NOT(p_tyNtParamCurr.bProjMagHeightChkPrep);
	tyP0410MagSel.tyMagDet.tyBtnMagHeightChkEn.uiRtStat.0	:= NOT(p_tyNtParamCurr.bProjMagHeightChkPrep);
	tyP0410MagSel.tyMagSel.tyBitmapBrder.uiRtStat.0			:= NOT(p_tyNtParamCurr.bProjMagSafetyBarPrep OR p_tyNtParamCurr.bProjMagHeightChkPrep);

END_ACTION
```

#### Act_Main_P0800.st
```iecst
ACTION Act_Main_P0800:

	//Display
	tyP0800MagInfo.tyMagInfo2.tyLyr.uiRtStat.0	:= NOT(p_tyNtParamCurr.eProjMag = LDMagTriple OR p_tyNtParamCurr.eProjMag = LDMagQuadruple);

	IF p_tyNtParamCurr.eProjMag <> LDMagQuadruple THEN
		tyP0800MagInfo.tyMagInfo4.tyLyr.uiRtStat.0	:= TRUE;

	END_IF

	tyP0800MagInfo.tyMagInfo1.tyBtnMag1SetEmpty.uiRtStat.0 := p_tyNtParamCurr.bProjLifterMagPlatform;
	tyP0800MagInfo.tyMagInfo1.tyBtnMag2SetEmpty.uiRtStat.0 := p_tyNtParamCurr.bProjLifterMagPlatform;
	tyP0800MagInfo.tyMagInfo2.tyBtnMag3SetEmpty.uiRtStat.0 := p_tyNtParamCurr.bProjLifterMagPlatform;

	tyP0800MagInfo.tyMagInfo1.tyBtnMag1SetEmpty.uiMaskRtStat.0 := p_tyNtParamCurr.bProjLifterMagPlatform;
	tyP0800MagInfo.tyMagInfo1.tyBtnMag2SetEmpty.uiMaskRtStat.0 := p_tyNtParamCurr.bProjLifterMagPlatform;
	tyP0800MagInfo.tyMagInfo2.tyBtnMag3SetEmpty.uiMaskRtStat.0 := p_tyNtParamCurr.bProjLifterMagPlatform;

END_ACTION
```

#### Act_Main_P0900.st
```iecst
ACTION Act_Main_P0900:

	//Display
	tyP0900GenIn.tyGenIn2.tyLyr.uiRtStat.0	:= NOT p_tyNtParamCurr.bProjMagOrientChkSenPrep;

	tyP0900GenIn.tyGenIn1.tyBtnLifterTimingBeltSen.uiRtStat.0	:= p_tyNtParamCurr.tyDISettings.diLifterTimingBeltSen = 0;
	tyP0900GenIn.tyGenIn1.tyBtnLifterSafetyLmtSW1.uiRtStat.0	:= p_tyNtParamCurr.tyDISettings.diLifterSafetyLmtSW1 = 0;
	tyP0900GenIn.tyGenIn1.tyBtnLifterSafetyLmtSW2.uiRtStat.0	:= p_tyNtParamCurr.tyDISettings.diLifterSafetyLmtSW2 = 0;
	tyP0900GenIn.tyGenIn1.tyBtnMag3PresentSen.uiRtStat.0		:= NOT(p_tyNtParamCurr.eProjMag = LDMagTriple OR p_tyNtParamCurr.eProjMag = LDMagQuadruple);
	tyP0900GenIn.tyGenIn1.tyBtnMag4PresentSen.uiRtStat.0		:= NOT(p_tyNtParamCurr.eProjMag = LDMagQuadruple);
	tyP0900GenIn.tyGenIn1.tyBtnCurtainSafetyRly.uiRtStat.0		:= p_tyNtParamCurr.tyDISettings.diCurtainSafetySig2 = 0;
	tyP0900GenIn.tyGenIn1.tyBtnMagWidthChk.uiRtStat.0		:= p_tyNtParamCurr.tyDISettings.diMagWidthChkSen = 0;

	tyP0900GenIn.tyGenIn2.tyBtnMag3OrientationChkSen1.uiRtStat.0	:= NOT(p_tyNtParamCurr.eProjMag = LDMagTriple);
	tyP0900GenIn.tyGenIn2.tyBtnMag3OrientationChkSen2.uiRtStat.0	:= NOT(p_tyNtParamCurr.eProjMag = LDMagTriple);

	tyP0900GenIn.tyGenIn2.tyBtnMag4OrientationChkSen1.uiRtStat.0	:= NOT(p_tyNtParamCurr.eProjMag = LDMagQuadruple);
	tyP0900GenIn.tyGenIn2.tyBtnMag4OrientationChkSen2.uiRtStat.0	:= NOT(p_tyNtParamCurr.eProjMag = LDMagQuadruple);

	tyP0900GenIn.tyGenIn2.tyBtnMag1OrientationChkSen2.uiRtStat	  := p_tyNtParamCurr.tyDISettings.diMag1OrientChkSen2 = 0;

END_ACTION
```

#### Act_Main_P0910.st
```iecst
ACTION Act_Main_P0910:

	//Display
	tyP0910GenOut.tyGenOut.tyBtnBuzzer.uiRtStat.0	:= p_tyNtParamCurr.tyDOSettings.diBuzzer = 0;
	tyP0910GenOut.tyGenOutCurtainSen.tyLyr.uiRtStat.0	:= NOT p_tyNtParamCurr.bProjCurtainSenPrep;

	tyP0910GenOut.tyGenOut.tyBtnTLRed.uiRtStat := p_tyNtParamCurr.eCustomerReq = Siemens;
	IF p_tyNtParamCurr.eCustomerReq = Siemens THEN
		tyP0910GenOut.tyGenOut.tyBtnTLAmber.usiTxtIdx := 2;
	ELSE
		tyP0910GenOut.tyGenOut.tyBtnTLAmber.usiTxtIdx := 0;
	END_IF

END_ACTION
```

#### Act_Main_P0920.st
```iecst
ACTION Act_Main_P0920:

	//Machine Bitmap//51 lifter 52 Trav 50 aw 53 puller conv 55 magconv 152 puller aw ;54 shutter 55safe bar
	IF p_tyNtParamCurr.eProjMag = LDMagTriple AND p_tyNtParamCurr.bProjLifterMagPlatform THEN
		tyP0920MtrNPneuCtrl.tyMtrNPneuCtrl.tyBtnAW.uiBitmapIdx				:= 301; //351
		tyP0920MtrNPneuCtrl.tyMtrNPneuCtrl.tyBtnLifter.uiBitmapIdx			:= 408-51;
		tyP0920MtrNPneuCtrl.tyMtrNPneuCtrl.tyBtnTrav.uiBitmapIdx			:= 409-52;
		tyP0920MtrNPneuCtrl.tyMtrNPneuCtrl.tyBtnPullerConv.uiBitmapIdx		:= 297;
		tyP0920MtrNPneuCtrl.tyMtrNPneuCtrl.tyBtnMag1Conv.uiBitmapIdx		:= 100;
		tyP0920MtrNPneuCtrl.tyMtrNPneuCtrl.tyBtnMag2Conv.uiBitmapIdx		:= 100;
		tyP0920MtrNPneuCtrl.tyMtrNPneuCtrl.tyBtnMag3Conv.uiBitmapIdx		:= 100;
		tyP0920MtrNPneuCtrl.tyMtrNPneuCtrlPneu.tyBtnShutter.uiBitmapIdx		:= 410-54;
		tyP0920MtrNPneuCtrl.tyMtrNPneuCtrlPneu.tyBtnSafetyBar.uiBitmapIdx	:= 100;
		tyP0920MtrNPneuCtrl.tyMtrNPneuCtrl.tyBtnAWPushPul.uiBitmapIdx		:= 200;

	ELSIF p_tyNtParamCurr.eProjMag = LDMagTriple AND p_tyNtParamCurr.bMagAutoVerifyPrep = FALSE THEN
		tyP0920MtrNPneuCtrl.tyMtrNPneuCtrl.tyBtnAW.uiBitmapIdx				:= 301;
		tyP0920MtrNPneuCtrl.tyMtrNPneuCtrl.tyBtnLifter.uiBitmapIdx			:= 100;
		tyP0920MtrNPneuCtrl.tyMtrNPneuCtrl.tyBtnTrav.uiBitmapIdx			:= 100;
		tyP0920MtrNPneuCtrl.tyMtrNPneuCtrl.tyBtnPullerConv.uiBitmapIdx		:= 297;
		tyP0920MtrNPneuCtrl.tyMtrNPneuCtrl.tyBtnMag1Conv.uiBitmapIdx		:= 100;
		tyP0920MtrNPneuCtrl.tyMtrNPneuCtrl.tyBtnMag2Conv.uiBitmapIdx		:= 100;
		tyP0920MtrNPneuCtrl.tyMtrNPneuCtrl.tyBtnMag3Conv.uiBitmapIdx		:= 100;
		tyP0920MtrNPneuCtrl.tyMtrNPneuCtrlPneu.tyBtnShutter.uiBitmapIdx		:= 100;
		tyP0920MtrNPneuCtrl.tyMtrNPneuCtrlPneu.tyBtnSafetyBar.uiBitmapIdx	:= 100;
		tyP0920MtrNPneuCtrl.tyMtrNPneuCtrl.tyBtnAWPushPul.uiBitmapIdx		:= 200;
	ELSIF p_tyNtParamCurr.eProjMag = LDMagTriple AND p_tyNtParamCurr.bMagAutoVerifyPrep = TRUE THEN
		tyP0920MtrNPneuCtrl.tyMtrNPneuCtrl.tyBtnAW.uiBitmapIdx				:= 200;
		tyP0920MtrNPneuCtrl.tyMtrNPneuCtrl.tyBtnLifter.uiBitmapIdx			:= 4;
		tyP0920MtrNPneuCtrl.tyMtrNPneuCtrl.tyBtnTrav.uiBitmapIdx			:= 4;
		tyP0920MtrNPneuCtrl.tyMtrNPneuCtrl.tyBtnPullerConv.uiBitmapIdx		:= 200;
		tyP0920MtrNPneuCtrl.tyMtrNPneuCtrl.tyBtnMag1Conv.uiBitmapIdx		:= 2;
		tyP0920MtrNPneuCtrl.tyMtrNPneuCtrl.tyBtnMag2Conv.uiBitmapIdx		:= 2;
		tyP0920MtrNPneuCtrl.tyMtrNPneuCtrl.tyBtnMag3Conv.uiBitmapIdx		:= 2;
		tyP0920MtrNPneuCtrl.tyMtrNPneuCtrlPneu.tyBtnShutter.uiBitmapIdx		:= 6;
		tyP0920MtrNPneuCtrl.tyMtrNPneuCtrlPneu.tyBtnSafetyBar.uiBitmapIdx	:= 0;
		tyP0920MtrNPneuCtrl.tyMtrNPneuCtrl.tyBtnAWPushPul.uiBitmapIdx		:= 0;
	ELSIF p_tyNtParamCurr.eProjMag = LDMagDual AND p_tyNtParamCurr.bMagAutoVerifyPrep = TRUE THEN
		tyP0920MtrNPneuCtrl.tyMtrNPneuCtrl.tyBtnAW.uiBitmapIdx				:= 200;
		tyP0920MtrNPneuCtrl.tyMtrNPneuCtrl.tyBtnLifter.uiBitmapIdx			:= 200;
		tyP0920MtrNPneuCtrl.tyMtrNPneuCtrl.tyBtnTrav.uiBitmapIdx			:= 200;
		tyP0920MtrNPneuCtrl.tyMtrNPneuCtrl.tyBtnPullerConv.uiBitmapIdx		:= 200;
		tyP0920MtrNPneuCtrl.tyMtrNPneuCtrl.tyBtnMag1Conv.uiBitmapIdx		:= 200;
		tyP0920MtrNPneuCtrl.tyMtrNPneuCtrl.tyBtnMag2Conv.uiBitmapIdx		:= 200;
		tyP0920MtrNPneuCtrl.tyMtrNPneuCtrl.tyBtnMag3Conv.uiBitmapIdx		:= 200;
		tyP0920MtrNPneuCtrl.tyMtrNPneuCtrlPneu.tyBtnShutter.uiBitmapIdx		:= 200;
		tyP0920MtrNPneuCtrl.tyMtrNPneuCtrlPneu.tyBtnSafetyBar.uiBitmapIdx	:= 0;
		tyP0920MtrNPneuCtrl.tyMtrNPneuCtrl.tyBtnAWPushPul.uiBitmapIdx		:= 0;
	ELSIF p_tyNtParamCurr.eProjMag = LDMagQuadruple AND p_tyNtParamCurr.bMagAutoVerifyPrep = TRUE THEN
		tyP0920MtrNPneuCtrl.tyMtrNPneuCtrl.tyBtnAW.uiBitmapIdx				:= 200;
		tyP0920MtrNPneuCtrl.tyMtrNPneuCtrl.tyBtnLifter.uiBitmapIdx			:= 16;
		tyP0920MtrNPneuCtrl.tyMtrNPneuCtrl.tyBtnTrav.uiBitmapIdx			:= 16;
		tyP0920MtrNPneuCtrl.tyMtrNPneuCtrl.tyBtnPullerConv.uiBitmapIdx		:= 200;
		tyP0920MtrNPneuCtrl.tyMtrNPneuCtrl.tyBtnMag1Conv.uiBitmapIdx		:= 6;
		tyP0920MtrNPneuCtrl.tyMtrNPneuCtrl.tyBtnMag2Conv.uiBitmapIdx		:= 200;
		tyP0920MtrNPneuCtrl.tyMtrNPneuCtrl.tyBtnMag3Conv.uiBitmapIdx		:= 200;
		tyP0920MtrNPneuCtrl.tyMtrNPneuCtrlPneu.tyBtnShutter.uiBitmapIdx		:= 8;
		tyP0920MtrNPneuCtrl.tyMtrNPneuCtrlPneu.tyBtnSafetyBar.uiBitmapIdx	:= 0;
		tyP0920MtrNPneuCtrl.tyMtrNPneuCtrl.tyBtnAWPushPul.uiBitmapIdx		:= 0;
	ELSIF p_tyNtParamCurr.eProjMag = LDMagDual AND p_tyNtParamCurr.bMagAutoVerifyPrep = FALSE THEN
		tyP0920MtrNPneuCtrl.tyMtrNPneuCtrl.tyBtnAW.uiBitmapIdx				:= 200;
		tyP0920MtrNPneuCtrl.tyMtrNPneuCtrl.tyBtnLifter.uiBitmapIdx			:= 200;
		tyP0920MtrNPneuCtrl.tyMtrNPneuCtrl.tyBtnTrav.uiBitmapIdx			:= 200;
		tyP0920MtrNPneuCtrl.tyMtrNPneuCtrl.tyBtnPullerConv.uiBitmapIdx		:= 200;
		tyP0920MtrNPneuCtrl.tyMtrNPneuCtrl.tyBtnMag1Conv.uiBitmapIdx		:= 200;
		tyP0920MtrNPneuCtrl.tyMtrNPneuCtrl.tyBtnMag2Conv.uiBitmapIdx		:= 200;
		tyP0920MtrNPneuCtrl.tyMtrNPneuCtrl.tyBtnMag3Conv.uiBitmapIdx		:= 200;
		tyP0920MtrNPneuCtrl.tyMtrNPneuCtrlPneu.tyBtnShutter.uiBitmapIdx		:= 200;
		tyP0920MtrNPneuCtrl.tyMtrNPneuCtrlPneu.tyBtnSafetyBar.uiBitmapIdx	:= 0;
		tyP0920MtrNPneuCtrl.tyMtrNPneuCtrl.tyBtnAWPushPul.uiBitmapIdx		:= 0;

	ELSE
		tyP0920MtrNPneuCtrl.tyMtrNPneuCtrl.tyBtnAW.uiBitmapIdx				:= 0;
		tyP0920MtrNPneuCtrl.tyMtrNPneuCtrl.tyBtnLifter.uiBitmapIdx			:= 0;
		tyP0920MtrNPneuCtrl.tyMtrNPneuCtrl.tyBtnTrav.uiBitmapIdx			:= 0;
		tyP0920MtrNPneuCtrl.tyMtrNPneuCtrl.tyBtnPullerConv.uiBitmapIdx		:= 0;
		tyP0920MtrNPneuCtrl.tyMtrNPneuCtrl.tyBtnMag1Conv.uiBitmapIdx		:= 0;
		tyP0920MtrNPneuCtrl.tyMtrNPneuCtrl.tyBtnMag2Conv.uiBitmapIdx		:= 0;
		tyP0920MtrNPneuCtrl.tyMtrNPneuCtrl.tyBtnMag3Conv.uiBitmapIdx		:= 0;
		tyP0920MtrNPneuCtrl.tyMtrNPneuCtrlPneu.tyBtnShutter.uiBitmapIdx		:= 0;
		tyP0920MtrNPneuCtrl.tyMtrNPneuCtrlPneu.tyBtnSafetyBar.uiBitmapIdx	:= 0;
		tyP0920MtrNPneuCtrl.tyMtrNPneuCtrl.tyBtnAWPushPul.uiBitmapIdx		:= 0;
	END_IF

	//Auto Width
	tyP0920MtrNPneuCtrl.tyMtrNPneuCtrl.tyBtnAW.uiRtStat.0	:= NOT p_tyNtParamCurr.bAWPrep;

	//Pusher Auto Width
	tyP0920MtrNPneuCtrl.tyMtrNPneuCtrl.tyBtnAWPushPul.uiRtStat.0	:= NOT p_tyNtParamCurr.bAWPusherPrep;

	//Pneumatic
	tyP0920MtrNPneuCtrl.tyMtrNPneuCtrlPneu.tyLyr.uiRtStat.0	:= NOT(p_tyNtParamCurr.bProjInletShutPrep OR p_tyNtParamCurr.bProjOutletShutPrep);

	//Shutter
	tyP0920MtrNPneuCtrl.tyMtrNPneuCtrlPneu.tyBtnShutter.uiRtStat.0  := NOT(p_tyNtParamCurr.bProjInletShutPrep OR p_tyNtParamCurr.bProjOutletShutPrep);

	//Magazine Conveyor
	tyP0920MtrNPneuCtrl.tyMtrNPneuCtrl.tyBtnMag1Conv.uiRtStat.0	:= NOT (p_tyNtParamCurr.bProjMag1ConvPrep OR p_tyNtParamCurr.bProjMag2ConvPrep OR p_tyNtParamCurr.bProjMag3ConvPrep) OR p_tyNtParamCurr.bProjLifTravMnlLoad ;
//	tyP0920MtrNPneuCtrl.tyMtrNPneuCtrl.tyBtnMag2Conv.uiRtStat.0	:= NOT p_tyNtParamCurr.bProjMag2ConvPrep;
//	tyP0920MtrNPneuCtrl.tyMtrNPneuCtrl.tyBtnMag3Conv.uiRtStat.0	:= NOT(p_tyNtParamCurr.bProjMag3ConvPrep AND (p_tyNtParamCurr.eProjMag = LDMagTriple));

	//Safety Bar
	tyP0920MtrNPneuCtrl.tyMtrNPneuCtrlPneu.tyBtnSafetyBar.uiRtStat.0	:= NOT p_tyNtParamCurr.bProjMagSafetyBarPrep;
	//TrolleyLck
	tyP0920MtrNPneuCtrl.tyMtrNPneuCtrlPneu.tyBtnTrolleyLck.uiRtStat.0	:= NOT p_tyNtParamCurr.bProjTrolleyLckPrep;

END_ACTION
```

#### Act_Main_P0921.st
```iecst
ACTION Act_Main_P0921:
	//Title
	IF p_tyNtParamCurr.bProjShutter2Prep THEN  //>1 inlet shutter
		tyP0921InletNOutletShutter.tyInletShutterCom.tyTxtTit.usiValueIdx := 145-5;
	ELSE
		tyP0921InletNOutletShutter.tyInletShutterCom.tyTxtTit.usiValueIdx := 0;//
	END_IF
	IF p_tyNtParamCurr.bProjOutShutter2Prep THEN
		tyP0921InletNOutletShutter.tyOutletShutterCom.tyTxtTit.usiValueIdx := 148-6;
	ELSE
		tyP0921InletNOutletShutter.tyOutletShutterCom.tyTxtTit.usiValueIdx := 0;
	END_IF

	//Display
	tyP0921InletNOutletShutter.tyInletShutterCom.tyLyr.uiRtStat.0	:= NOT(p_tyNtParamCurr.bProjInletShutPrep);
	tyP0921InletNOutletShutter.tyInletShutterDC.tyLyr.uiRtStat.0	:= TRUE;
	tyP0921InletNOutletShutter.tyInletShutterFB.tyLyr.uiRtStat.0	:= NOT(p_tyNtParamCurr.bProjInletShutPrep);

	tyP0921InletNOutletShutter.tyOutletShutterCom.tyLyr.uiRtStat.0	:= NOT(p_tyNtParamCurr.bProjOutletShutPrep);
	tyP0921InletNOutletShutter.tyOutletShutterDC.tyLyr.uiRtStat.0	:= TRUE;
	tyP0921InletNOutletShutter.tyOutletShutterFB.tyLyr.uiRtStat.0	:= NOT(p_tyNtParamCurr.bProjOutletShutPrep);

	//Inlet shutter 2,3_ opening
	tyP0921InletNOutletShutter.tyInletShutterFB.tyBtnOpen2.uiRtStat :=  TRUE;
	tyP0921InletNOutletShutter.tyInletShutterFB.tyBtnOpen3.uiRtStat :=  TRUE;
	tyP0921InletNOutletShutter.tyInletShutterDC.tyBtnOpen2.uiRtStat :=  TRUE;
	tyP0921InletNOutletShutter.tyInletShutterDC.tyBtnOpen3.uiRtStat :=  TRUE;

END_ACTION
```

#### Act_Main_P0923.st
```iecst
ACTION Act_Main_P0923:

END_ACTION
```

#### Act_Main_P0930.st
```iecst
ACTION Act_Main_P0930:

	//Display
	tyP0930MagConv1.tyCom.tyBtnMagAIVPosSen1.uiRtStat.0			:= p_tyNtParamCurr.tyDISettings.diMag1AGVInPosSen1 = 0;
	tyP0930MagConv1.tyCom.tyBtnMagAIVPosSen2.uiRtStat.0			:= p_tyNtParamCurr.tyDISettings.diMag1AGVInPosSen2 = 0;
	tyP0930MagConv1.tyCom.tyBtnMagOrientationChkSen1.uiRtStat.0	:= p_tyNtParamCurr.tyDISettings.diMag1OrientChkSen1 = 0;
	tyP0930MagConv1.tyCom.tyBtnMagOrientationChkSen2.uiRtStat.0	:= p_tyNtParamCurr.tyDISettings.diMag1OrientChkSen2 = 0;

	tyP0930MagConv1.tyCom.tyBtnRemoteClampRS.uiRtStat.0			:= TRUE;
	tyP0930MagConv1.tyCom.tyBtnRemoteUnclampRS.uiRtStat.0		:= p_tyNtParamCurr.tyDISettings.diMag1RemoteUnclampRS = 0;
	tyP0930MagConv1.tyCom.tyBtnFixedClampRS.uiRtStat.0			:= p_tyNtParamCurr.bMagAutoVerifyPrep;

	tyP0930MagConv1.tyCom.tyBtnHeightSen.uiRtStat.0				:= NOT (p_tyNtParamCurr.bMagAutoVerifyPrep OR p_tyNtParamCurr.bProjMagHeightChkPrep);
	tyP0930MagConv1.tyCom.tyBtnCAB717Sen.uiRtStat.0				:= NOT p_tyNtParamCurr.bMagAutoVerifyPrep;
	tyP0930MagConv1.tyCom.tyBtnMagLargeSen.uiRtStat.0			:= NOT p_tyNtParamCurr.bMagAutoVerifyPrep;
	tyP0930MagConv1.tyCom.tyBtnMagSmallSen.uiRtStat.0			:= NOT p_tyNtParamCurr.bMagAutoVerifyPrep;
	tyP0930MagConv1.tyCom.tyBtnSelClampRS.uiRtStat.0			:= NOT p_tyNtParamCurr.bMagAutoVerifyPrep;
	tyP0930MagConv1.tyCom.tyBtnSelUnclampRS.uiRtStat.0			:= NOT p_tyNtParamCurr.bMagAutoVerifyPrep;
	tyP0930MagConv1.tyCom.tyBtnSltLckSen.uiRtStat.0				:= p_tyNtParamCurr.tyDISettings.diSlotLckSenMag1 = 0;

	IF p_tyNtParamCurr.bMagAutoVerifyPrep = FALSE THEN
		tyP0930MagConv1.tyCom.tyBtnFixedClampRS.usiTxtIdx:=4;
		tyP0930MagConv1.tyCom.tyBtnFixedUnclampRS.usiTxtIdx:=4;
	ELSE
		tyP0930MagConv1.tyCom.tyBtnFixedClampRS.usiTxtIdx:=4;
		tyP0930MagConv1.tyCom.tyBtnFixedUnclampRS.usiTxtIdx:=4;
	END_IF

END_ACTION
```

#### Act_Main_P0931.st
```iecst
ACTION Act_Main_P0931:

	//Display
	tyP0931MagConv2.tyCom.tyBtnMagAIVPosSen1.uiRtStat.0			:= p_tyNtParamCurr.tyDISettings.diMag2AGVInPosSen1 = 0;
	tyP0931MagConv2.tyCom.tyBtnMagAIVPosSen2.uiRtStat.0			:= p_tyNtParamCurr.tyDISettings.diMag2AGVInPosSen2 = 0;
	tyP0931MagConv2.tyCom.tyBtnMagOrientationChkSen1.uiRtStat.0	:= p_tyNtParamCurr.tyDISettings.diMag2OrientChkSen1 = 0;
	tyP0931MagConv2.tyCom.tyBtnMagOrientationChkSen2.uiRtStat.0	:= p_tyNtParamCurr.tyDISettings.diMag2OrientChkSen2 = 0;

	tyP0931MagConv2.tyCom.tyBtnRemoteClampRS.uiRtStat.0			:= TRUE;
	tyP0931MagConv2.tyCom.tyBtnRemoteUnclampRS.uiRtStat.0		:= p_tyNtParamCurr.tyDISettings.diMag2RemoteUnclampRS = 0;
	tyP0931MagConv2.tyCom.tyBtnFixedClampRS.uiRtStat.0			:= p_tyNtParamCurr.bMagAutoVerifyPrep;

	tyP0931MagConv2.tyCom.tyBtnHeightSen.uiRtStat.0				:= NOT (p_tyNtParamCurr.bMagAutoVerifyPrep OR p_tyNtParamCurr.bProjMagHeightChkPrep);
	tyP0931MagConv2.tyCom.tyBtnCAB717Sen.uiRtStat.0				:= NOT p_tyNtParamCurr.bMagAutoVerifyPrep;
	tyP0931MagConv2.tyCom.tyBtnMagLargeSen.uiRtStat.0			:= NOT p_tyNtParamCurr.bMagAutoVerifyPrep;
	tyP0931MagConv2.tyCom.tyBtnMagSmallSen.uiRtStat.0			:= NOT p_tyNtParamCurr.bMagAutoVerifyPrep;
	tyP0931MagConv2.tyCom.tyBtnSelClampRS.uiRtStat.0			:= NOT p_tyNtParamCurr.bMagAutoVerifyPrep;
	tyP0931MagConv2.tyCom.tyBtnSelUnclampRS.uiRtStat.0			:= NOT p_tyNtParamCurr.bMagAutoVerifyPrep;
	tyP0931MagConv2.tyCom.tyBtnSltLckSen.uiRtStat.0				:= p_tyNtParamCurr.tyDISettings.diSlotLckSenMag2 = 0;

	IF p_tyNtParamCurr.bMagAutoVerifyPrep = FALSE THEN
		tyP0931MagConv2.tyCom.tyBtnFixedClampRS.usiTxtIdx:=4;
		tyP0931MagConv2.tyCom.tyBtnFixedUnclampRS.usiTxtIdx:=4;
	ELSE
		tyP0931MagConv2.tyCom.tyBtnFixedClampRS.usiTxtIdx:=4;
		tyP0931MagConv2.tyCom.tyBtnFixedUnclampRS.usiTxtIdx:=4;
	END_IF

END_ACTION
```

#### Act_Main_P0932.st
```iecst
ACTION Act_Main_P0932:

	//Display
	tyP0932MagConv3.tyCom.tyBtnMagAIVPosSen1.uiRtStat.0			:= p_tyNtParamCurr.tyDISettings.diMag3AGVInPosSen1 = 0;
	tyP0932MagConv3.tyCom.tyBtnMagAIVPosSen2.uiRtStat.0			:= p_tyNtParamCurr.tyDISettings.diMag3AGVInPosSen2 = 0;
	tyP0932MagConv3.tyCom.tyBtnMagOrientationChkSen1.uiRtStat.0	:= p_tyNtParamCurr.tyDISettings.diMag3OrientChkSen1 = 0;
	tyP0932MagConv3.tyCom.tyBtnMagOrientationChkSen2.uiRtStat.0	:= p_tyNtParamCurr.tyDISettings.diMag3OrientChkSen2 = 0;

	tyP0932MagConv3.tyCom.tyBtnRemoteClampRS.uiRtStat.0			:= TRUE;
	tyP0932MagConv3.tyCom.tyBtnRemoteUnclampRS.uiRtStat.0		:= p_tyNtParamCurr.tyDISettings.diMag3RemoteUnclampRS = 0;
	tyP0932MagConv3.tyCom.tyBtnFixedClampRS.uiRtStat.0			:= p_tyNtParamCurr.bMagAutoVerifyPrep;

	tyP0932MagConv3.tyCom.tyBtnHeightSen.uiRtStat.0				:= NOT (p_tyNtParamCurr.bMagAutoVerifyPrep OR p_tyNtParamCurr.bProjMagHeightChkPrep);
	tyP0932MagConv3.tyCom.tyBtnCAB717Sen.uiRtStat.0				:= NOT p_tyNtParamCurr.bMagAutoVerifyPrep;
	tyP0932MagConv3.tyCom.tyBtnMagLargeSen.uiRtStat.0			:= NOT p_tyNtParamCurr.bMagAutoVerifyPrep;
	tyP0932MagConv3.tyCom.tyBtnMagSmallSen.uiRtStat.0			:= NOT p_tyNtParamCurr.bMagAutoVerifyPrep;
	tyP0932MagConv3.tyCom.tyBtnSelClampRS.uiRtStat.0			:= NOT p_tyNtParamCurr.bMagAutoVerifyPrep;
	tyP0932MagConv3.tyCom.tyBtnSelUnclampRS.uiRtStat.0			:= NOT p_tyNtParamCurr.bMagAutoVerifyPrep;

	IF p_tyNtParamCurr.bMagAutoVerifyPrep = FALSE THEN
		tyP0932MagConv3.tyCom.tyBtnFixedClampRS.usiTxtIdx:=4;
		tyP0932MagConv3.tyCom.tyBtnFixedUnclampRS.usiTxtIdx:=4;
	ELSE
		tyP0932MagConv3.tyCom.tyBtnFixedClampRS.usiTxtIdx:=4;
		tyP0932MagConv3.tyCom.tyBtnFixedUnclampRS.usiTxtIdx:=4;
	END_IF

END_ACTION
```

#### Act_Main_P0933.st
```iecst
ACTION Act_Main_P0933:

	//Display
	tyP0933PullConv.tyCom.tyBtnRotHmRS.uiRtStat.0	:= NOT p_tyNtParamCurr.bProjPullerRotCylPrep;
	tyP0933PullConv.tyCom.tyBtnRotRmRS.uiRtStat.0	:= NOT p_tyNtParamCurr.bProjPullerRotCylPrep;

	tyP0933PullConv.tyCom.tyBtnExtSlwSen.uiRtStat.0	:= NOT p_tyNtParamCurr.bProjMotorizedPullerPrep;
	tyP0933PullConv.tyCom.tyBtnRetSlwSen.uiRtStat.0	:= NOT p_tyNtParamCurr.bProjMotorizedPullerPrep;
	tyP0933PullConv.tyCom.tyBtnAlarmSig.uiRtStat.0	:= NOT (p_tyNtParamCurr.bProjMotorizedPullerPrep AND NOT(p_tyNtParamCurr.bProjServoPullerPusherPrep));
	tyP0933PullConv.tyCom.tyBtnTorqueSig.uiRtStat.0	:= NOT (p_tyNtParamCurr.bProjMotorizedPullerPrep AND NOT(p_tyNtParamCurr.bProjServoPullerPusherPrep));
	tyP0933PullConv.tyCom.tyBtnAntiJamSen.uiRtStat.0 :=   p_tyNtParamCurr.tyDISettings.diPullerAntiJam = 0;

//	tyP0933PullConv.tyFB.tyBtnCylEnt.uiRtStat.0		:= NOT p_tyNtParamCurr.bProjPullerRotCylPrep;
	tyP0933PullConv.tyFB.tyBtnRotToHm.uiRtStat.0	:= NOT p_tyNtParamCurr.bProjPullerRotCylPrep;
	tyP0933PullConv.tyFB.tyBtnRotToRm.uiRtStat.0	:= NOT p_tyNtParamCurr.bProjPullerRotCylPrep;

	tyP0933PullConv.tyDC.tyBtnRotToHm.uiRtStat.0	:= NOT p_tyNtParamCurr.bProjPullerRotCylPrep;
	tyP0933PullConv.tyDC.tyBtnRotToRm.uiRtStat.0	:= NOT p_tyNtParamCurr.bProjPullerRotCylPrep;

	tyP0933PullConv.tyFB.tyNumExtSpd.uiRtStat.0			:= NOT p_tyNtParamCurr.bProjMotorizedPullerPrep;
	tyP0933PullConv.tyFB.tyNumExtTorqPercent.uiRtStat.0	:= NOT p_tyNtParamCurr.bProjMotorizedPullerPrep;

	tyP0933PullConv.tyDC.tyBtnSpdBinBit0.uiRtStat.0	:=  NOT p_tyNtParamCurr.bProjMotorizedPullerPrep;
	tyP0933PullConv.tyDC.tyBtnSpdBinBit1.uiRtStat.0	:=  NOT p_tyNtParamCurr.bProjMotorizedPullerPrep;
	tyP0933PullConv.tyDC.tyBtnSpdBinBit2.uiRtStat.0	:=  NOT p_tyNtParamCurr.bProjMotorizedPullerPrep;

	tyP0933PullConv.tyDC.tyBtnSigOn.uiRtStat.0	:=  NOT p_tyNtParamCurr.bProjMotorizedPullerPrep;
	tyP0933PullConv.tyDC.tyBtnAlarmRst.uiRtStat.0:=  NOT p_tyNtParamCurr.bProjMotorizedPullerPrep;

	//Display
	tyP0933PullConv.tyFB.tyNumExtSpd.diValueMin	:= p_tyNtParamCurr.tyProdRcpMtrPshrExtSpd.diMin;
	tyP0933PullConv.tyFB.tyNumExtSpd.diValueMax	:= p_tyNtParamCurr.tyProdRcpMtrPshrExtSpd.diMax;

	tyP0933PullConv.tyFB.tyNumExtTorqPercent.diValueMin	:= p_tyNtParamCurr.tyProdRcpMtrPshrExtTorq.diMin;
	tyP0933PullConv.tyFB.tyNumExtTorqPercent.diValueMax	:= p_tyNtParamCurr.tyProdRcpMtrPshrExtTorq.diMax;

	tyP0933PullConv.tyCom.tyBtnConvClrSen.uiRtStat.0	:=  p_tyNtParamCurr.tyDISettings.diConvClrSen =0;

END_ACTION
```

#### Act_Main_P0935.st
```iecst
ACTION Act_Main_P0935:

	tyP0935Lifter.tyLifter.tyBtnGoLaneB.uiRtStat.0	:= NOT p_tyNtParamCurr.bProjLaneBPrep;

	//Display
	tyP0935Lifter.tyMotionStd.tyNumTargetPos.diValue	:= 0;
	tyP0935Lifter.tyMotionStd.tyNumStepSize.diValue		:= 0;
	tyP0935Lifter.tyMotionStd.tyNumNomSpd.diValue		:= (p_tyNtParamCurr.tyUILifterNomSpd.diMax + p_tyNtParamCurr.tyUILifterNomSpd.diMin) / 2;
	tyP0935Lifter.tyMotionStd.tyNumSlwSpd.diValue		:= (p_tyNtParamCurr.tyUILifterSlwSpd.diMax + p_tyNtParamCurr.tyUILifterSlwSpd.diMin) / 3;

	tyP0935Lifter.tyMotionStd.tyNumTargetPos.diValueMax	:= p_tyNtParamCurr.tyUILifterTargetPos.diMax;
	tyP0935Lifter.tyMotionStd.tyNumTargetPos.diValueMin	:= p_tyNtParamCurr.tyUILifterTargetPos.diMin;

	tyP0935Lifter.tyMotionStd.tyNumStepSize.diValueMax	:= p_tyNtParamCurr.tyUILifterStepSize.diMax;
	tyP0935Lifter.tyMotionStd.tyNumStepSize.diValueMin	:= p_tyNtParamCurr.tyUILifterStepSize.diMin;

	tyP0935Lifter.tyMotionStd.tyNumNomSpd.diValueMax	:= p_tyNtParamCurr.tyUILifterNomSpd.diMax;
	tyP0935Lifter.tyMotionStd.tyNumNomSpd.diValueMin	:= p_tyNtParamCurr.tyUILifterNomSpd.diMin;

	tyP0935Lifter.tyMotionStd.tyNumSlwSpd.diValueMax	:= p_tyNtParamCurr.tyUILifterSlwSpd.diMax;
	tyP0935Lifter.tyMotionStd.tyNumSlwSpd.diValueMin	:= p_tyNtParamCurr.tyUILifterSlwSpd.diMin;

	tyP0935Lifter.tyLifter.tyNumMagPos.diValue			:= 1;
	tyP0935Lifter.tyLifter.tyNumMagPos.diValueMin		:= 1;

	CASE p_tyNtParamCurr.eProjMag OF

		LDMagDual:
			tyP0935Lifter.tyLifter.tyNumMagPos.diValueMax		:= 2;

		LDMagTriple:
			tyP0935Lifter.tyLifter.tyNumMagPos.diValueMax		:= 3;

		LDMagQuadruple:
			tyP0935Lifter.tyLifter.tyNumMagPos.diValueMax		:= 4;

	END_CASE

END_ACTION
```

#### Act_Main_P0936.st
```iecst
ACTION Act_Main_P0936:

	//Display
	tyP0936Trav.tyTrav.tyBtnGoToLaneB.uiRtStat.0	:= NOT p_tyNtParamCurr.bProjLaneBPrep;
	tyP0936Trav.tyTrav.tyBtnGoToMag3.uiRtStat.0		:= NOT(p_tyNtParamCurr.eProjMag = LDMagTriple OR p_tyNtParamCurr.eProjMag = LDMagQuadruple);
	tyP0936Trav.tyTrav.tyBtnGoToMag4.uiRtStat.0		:= NOT(p_tyNtParamCurr.eProjMag = LDMagQuadruple);

	tyP0936Trav.tyMotionStd.tyNumTargetPos.diValue		:= 0;
	tyP0936Trav.tyMotionStd.tyNumStepSize.diValue		:= 0;
	tyP0936Trav.tyMotionStd.tyNumNomSpd.diValue			:= (p_tyNtParamCurr.tyUITravNomSpd.diMax + p_tyNtParamCurr.tyUITravNomSpd.diMin) / 2;
	tyP0936Trav.tyMotionStd.tyNumSlwSpd.diValue			:= (p_tyNtParamCurr.tyUITravSlwSpd.diMax + p_tyNtParamCurr.tyUITravSlwSpd.diMin) / 3;

	tyP0936Trav.tyMotionStd.tyNumTargetPos.diValueMax	:= p_tyNtParamCurr.tyUITravTargetPos.diMax;
	tyP0936Trav.tyMotionStd.tyNumTargetPos.diValueMin	:= p_tyNtParamCurr.tyUITravTargetPos.diMin;

	tyP0936Trav.tyMotionStd.tyNumStepSize.diValueMax	:= p_tyNtParamCurr.tyUITravStepSize.diMax;
	tyP0936Trav.tyMotionStd.tyNumStepSize.diValueMin	:= p_tyNtParamCurr.tyUITravStepSize.diMin;

	tyP0936Trav.tyMotionStd.tyNumNomSpd.diValueMax		:= p_tyNtParamCurr.tyUITravNomSpd.diMax;
	tyP0936Trav.tyMotionStd.tyNumNomSpd.diValueMin		:= p_tyNtParamCurr.tyUITravNomSpd.diMin;

	tyP0936Trav.tyMotionStd.tyNumSlwSpd.diValueMax		:= p_tyNtParamCurr.tyUITravSlwSpd.diMax;
	tyP0936Trav.tyMotionStd.tyNumSlwSpd.diValueMin		:= p_tyNtParamCurr.tyUITravSlwSpd.diMin;

END_ACTION
```

#### Act_Main_P0939.st
```iecst
ACTION Act_Main_P0939:

	//Display
	tyP0939MagConv4.tyCom.tyBtnMagAIVPosSen1.uiRtStat.0			:= p_tyNtParamCurr.tyDISettings.diMag4AGVInPosSen1 = 0;
	tyP0939MagConv4.tyCom.tyBtnMagAIVPosSen2.uiRtStat.0			:= p_tyNtParamCurr.tyDISettings.diMag4AGVInPosSen2 = 0;
	tyP0939MagConv4.tyCom.tyBtnMagOrientationChkSen1.uiRtStat.0	:= p_tyNtParamCurr.tyDISettings.diMag4OrientChkSen1 = 0;
	tyP0939MagConv4.tyCom.tyBtnMagOrientationChkSen2.uiRtStat.0	:= p_tyNtParamCurr.tyDISettings.diMag4OrientChkSen2 = 0;

	tyP0939MagConv4.tyCom.tyBtnRemoteClampRS.uiRtStat.0			:= TRUE;
	tyP0939MagConv4.tyCom.tyBtnRemoteUnclampRS.uiRtStat.0		:= p_tyNtParamCurr.tyDISettings.diMag4RemoteUnclampRS = 0;
	tyP0939MagConv4.tyCom.tyBtnFixedClampRS.uiRtStat.0			:= p_tyNtParamCurr.bMagAutoVerifyPrep;

	tyP0939MagConv4.tyCom.tyBtnHeightSen.uiRtStat.0				:= NOT p_tyNtParamCurr.bMagAutoVerifyPrep;
	tyP0939MagConv4.tyCom.tyBtnCAB717Sen.uiRtStat.0				:= NOT p_tyNtParamCurr.bMagAutoVerifyPrep;
	tyP0939MagConv4.tyCom.tyBtnMagLargeSen.uiRtStat.0			:= NOT p_tyNtParamCurr.bMagAutoVerifyPrep;
	tyP0939MagConv4.tyCom.tyBtnMagSmallSen.uiRtStat.0			:= NOT p_tyNtParamCurr.bMagAutoVerifyPrep;
	tyP0939MagConv4.tyCom.tyBtnSelClampRS.uiRtStat.0			:= NOT p_tyNtParamCurr.bMagAutoVerifyPrep;
	tyP0939MagConv4.tyCom.tyBtnSelUnclampRS.uiRtStat.0			:= NOT p_tyNtParamCurr.bMagAutoVerifyPrep;

	IF p_tyNtParamCurr.bMagAutoVerifyPrep = FALSE THEN
		tyP0939MagConv4.tyCom.tyBtnFixedClampRS.usiTxtIdx:=4;
		tyP0939MagConv4.tyCom.tyBtnFixedUnclampRS.usiTxtIdx:=4;
	ELSE
		tyP0939MagConv4.tyCom.tyBtnFixedClampRS.usiTxtIdx:=4;
		tyP0939MagConv4.tyCom.tyBtnFixedUnclampRS.usiTxtIdx:=4;
	END_IF

END_ACTION
```

#### Act_Main_P0940.st
```iecst
ACTION Act_Main_P0940:

	//Display
	tyP0940CommCtrl.tyDSSMEMAB.tyLyr.uiRtStat.0	:= NOT(p_tyNtParamCurr.bProjLaneBPrep);

	IF  p_tyNtParamCurr.bProjAGVPrep THEN

		tyP0940CommCtrl.tySOT.tySOTLyr1.uiRtStat.0 := FALSE;
		tyP0940CommCtrl.tySOT.tySOTLyr2.uiRtStat.0 := FALSE;
		tyP0940CommCtrl.tySOT.tySOTLyr3.uiRtStat.0 := p_tyNtParamCurr.eProjMag <> LDMagTriple AND p_tyNtParamCurr.eProjMag <> LDMagQuadruple;
		tyP0940CommCtrl.tySOT.tySOTLyr4.uiRtStat.0 := p_tyNtParamCurr.eProjMag <> LDMagQuadruple;

	ELSE

		tyP0940CommCtrl.tySOT.tySOTLyr1.uiRtStat.0 := TRUE;
		tyP0940CommCtrl.tySOT.tySOTLyr2.uiRtStat.0 := TRUE;
		tyP0940CommCtrl.tySOT.tySOTLyr3.uiRtStat.0 := TRUE;
		tyP0940CommCtrl.tySOT.tySOTLyr4.uiRtStat.0 := TRUE;

	END_IF

	tyP0940CommCtrl.tySOT.tyBtnAIVRcv1.uiRtStat.0 := NOT(p_tyNtParamCurr.bProjSOTSensorPrep);
	tyP0940CommCtrl.tySOT.tyBtnAIVRcv2.uiRtStat.0 := NOT(p_tyNtParamCurr.bProjSOTSensorPrep);
	tyP0940CommCtrl.tySOT.tyBtnAIVRcv3.uiRtStat.0 := NOT(p_tyNtParamCurr.bProjSOTSensorPrep);
	tyP0940CommCtrl.tySOT.tyBtnAIVRcv4.uiRtStat.0 := NOT(p_tyNtParamCurr.bProjSOTSensorPrep);

	tyP0940CommCtrl.tySOT.tyBtnFleetMgrActive.uiRtStat.0 := NOT(p_tyNtParamCurr.bProjAGVPrep);
	tyP0940CommCtrl.tySOT.tyTxtAIVCommProtocol.uiRtStat.0 :=  NOT(p_tyNtParamCurr.bProjAGVPrep);

END_ACTION
```

#### Act_Main_P0950.st
```iecst
ACTION Act_Main_P0950:

	//Display
//	tyP0950Simu.tyAGVToMc.tyLyr.uiRtStat.0 := NOT(p_tyNtParamCurr.bProjAGVPrep AND p_tyMcParamCurr.bAGVComEn);
	tyP0950Simu.tySimu.tyLyr.uiRtStat.0 := TRUE;
	tyP0950Simu.tySimu.tyLyr1.uiRtStat.0 := NOT((p_tyNtParamCurr.bProjAGVPrep AND p_tyMcParamCurr.bAGVComEn) OR p_tyNtParamCurr.bProjInletShutPrep);
	tyP0950Simu.tySimu.tyLyrMag3.uiRtStat.0 := NOT(p_tyNtParamCurr.bProjAGVPrep AND p_tyMcParamCurr.bAGVComEn AND (p_tyNtParamCurr.eProjMag = LDMagTriple OR p_tyNtParamCurr.eProjMag = LDMagQuadruple));
	tyP0950Simu.tySimu.tyLyrMag4.uiRtStat.0 := NOT(p_tyNtParamCurr.bProjAGVPrep AND p_tyMcParamCurr.bAGVComEn AND p_tyNtParamCurr.eProjMag = LDMagQuadruple);

	IF p_tyNtParamCurr.eProjMag = LDMagDual THEN
		tyP0950Simu.tyAGVToMc.tyBtnAGV3Occupied.uiRtStat		:= TRUE;
		tyP0950Simu.tyAGVToMc.tyBtnAGVInPos3.uiRtStat   		:= TRUE;
		tyP0950Simu.tyMcToAGV.tyBtnMag3Auto.uiRtStat			:= TRUE;
		tyP0950Simu.tyMcToAGV.tyBtnMag3Empty.uiRtStat   		:= TRUE;
		tyP0950Simu.tyMcToAGV.tyBtnMag3IncorrectModel.uiRtStat 	:= TRUE;
		tyP0950Simu.tyMcToAGV.tyBtnMag3Occupied.uiRtStat 		:= TRUE;
		tyP0950Simu.tyMcToAGV.tyBtnMag3Rdy.uiRtStat				:= TRUE;
	END_IF
END_ACTION
```

#### Act_Main_P1020.st
```iecst
ACTION Act_Main_P1020:

	//Display
	tyP1020McSetNavi.tyNavi.tyBtnVCommSet.uiRtStat.0	:= NOT(p_tyNtParamCurr.bLFPrep OR p_tyNtParamCurr.bLCSLFPrep OR p_tyNtParamCurr.bLCSReqRcpPrep OR p_tyNtParamCurr.bLCSLiveDatPrep);
	tyP1020McSetNavi.tyNavi.tyBtnAIVCommSet.uiRtStat.0	:= TRUE;

	tyP1020McSetNavi.tyNavi.tyBtnUSBSet.uiRtStat.0		:= NOT(p_tyNtParamCurr.bUSBScannerPrep);
	tyP1020McSetNavi.tyNavi.tyBtnRS232Set.uiRtStat.0	:= NOT(p_tyNtParamCurr.bRS232ScannerPrep);

	//new for Hermes 1.3
	IF (p_tyNtParamCurr.bHermesSvyPrep AND p_tyMcParamCurr.bHermesSvyEn)
		OR p_tyNtParamCurr.bLFPrep OR p_tyNtParamCurr.bLCSLFPrep OR p_tyNtParamCurr.bLCSReqRcpPrep OR p_tyNtParamCurr.bLCSLiveDatPrep
		OR p_tyNtParamCurr.bLCSManageRcpPrep OR p_tyNtParamCurr.bLFUsrSetPrep OR p_tyNtParamCurr.bLFUsrSetPrep
		(*OR p_tyNtParamCurr.bUSWidthChkPrep*) OR p_tyNtParamCurr.bDSWidthChkPrep THEN

		fUIInRtStatOff(ADR(tyP1020McSetNavi.tyNavi.tyBtnVCommSet.uiRtStat));
	ELSE
		fUIInRtStatHide(ADR(tyP1020McSetNavi.tyNavi.tyBtnVCommSet.uiRtStat));
	END_IF
END_ACTION
```
